// TwinCAT 3 PLC project PRG_B_Base
// Title: B_Base
// Company: RafalOS
// Author: Rafał Osajda
// ProjectVersion: 0.0.0.59
// ProgramVersion: 3.1.4024.0
// libraries:
//   Tc2_Standard, * (Beckhoff Automation GmbH)
//   Tc2_System, * (Beckhoff Automation GmbH)
//   Tc2_Utilities, * (Beckhoff Automation GmbH)
//   Tc3_Module, * (Beckhoff Automation GmbH)
// project tree:
//   DUTs Events/ E_BaseEvents_Category.TcDUT (not stored), E_BaseEvents_Action.TcDUT, ST_BaseEvents.TcDUT, ST_BaseEvents_ActiveEvents.TcDUT, ST_BaseEvents_Definition.TcDUT, ST_BaseEvents_Queue.TcDUT, ST_BaseEvents_Memory.TcDUT, ST_BaseEvents_RowInQueue.TcDUT, ST_BaseEvents_RowInMemory.TcDUT, ST_BaseEvents_InformationAboutEventsForHMI.TcDUT
//   DUTs/ E_BaseElementType.TcDUT, E_BaseLocation.TcDUT, E_BaseMachineState.TcDUT, E_BaseMachineMode.TcDUT, ST_BaseCommonData.TcDUT (not stored), ST_BaseDescriptor.TcDUT (not stored), ST_BaseElementIdentifier.TcDUT, ST_BaseLocationDesctription.TcDUT, ST_BaseLabel.TcDUT
//   FUNs/ CreateElementCode.TcPOU
//   GVLs/ GVL_BaseConstans.TcGVL
//   ITFs/ ITF_DecoratedElement.TcIO
//   / PlcTask.TcTTO (not stored)
//   POUs Compilation/ PRG_Compilation.TcPOU
//   POUs/A01_Base/ ITF_Base.TcIO (not stored), FB_Base.TcPOU
//   POUs/A07_FB_BaseTopElement/ ITF_BaseSaM.TcIO, ITF_BaseSaMStateMethod.TcIO, FB_BaseTopElement.TcPOU, ITF_BaseTopElement.TcIO, ITF_BaseTopElement_HMI_Connector.TcIO
//   POUs/B01_Komunikator/ ITF_BaseCommunicator.TcIO, ITF_BaseMessengerRecipient.TcIO (not stored), ITF_BaseMessengerSender.TcIO, FB_BaseCommunicator.TcPOU, ST_BaseCommunicatorData.TcDUT (not stored), ST_BaseCommunicatorStack.TcDUT (not stored), ST_BaseCommunicatorMassege.TcDUT
//   POUs/B02_Recipes/ FB_BaseRecipe.TcPOU, ITF_BaseCreateTemplateOfRecipe.TcIO, ITF_BaseCreatingTemplateMethod.TcIO, ST_BaseRecipeListRow.TcDUT (not stored), ST_BaseRecipe.TcDUT
//   POUs/A00_Basic/ FB_BaseLabel.TcPOU, FB_BaseTime.TcPOU, FB_BaseCommand.TcPOU, FB_BaseDescriptor.TcPOU, FB_BaseFlag.TcPOU, FB_BaseImpulse.TcPOU, FB_BaseLocation.TcPOU, ITF_BaseDescriptor.TcIO, ITF_BaseFlag.TcIO, ITF_BaseFlagGet.TcIO (not stored), ITF_BaseFlagSet.TcIO, ITF_BaseImpulse.TcIO, ITF_BaseLabel.TcIO (not stored), ITF_BaseLocation.TcIO, ITF_BaseTime.TcIO
//   POUs/A02_FB_BaseLogger/ FB_BaseLogger.TcPOU, ITF_BaseLogger.TcIO, ITF_BaseLogger_HMI_Connector.TcIO, ITF_BaseLogger_Item.TcIO, ST_BaseLogger_ItemDataToDisplay.TcDUT
//   POUs/A03_FB_BaseLoggerElement/ FB_BaseLoggerElement.TcPOU, ITF_BaseLoggerElement.TcIO, ITF_BaseLoggerElement_HMI_Connector.TcIO
//   POUs/A04_FB_BaseComponent/ FB_BaseComponent.TcPOU, ITF_BaseComponent.TcIO, ITF_BaseComponent_HMI_Connector.TcIO, ST_Parameters.TcDUT (not stored)
//   POUs/A05_FB_BaseControlElement/ FB_BaseControlElement.TcPOU, ITF_BaseControlElement.TcIO, ITF_BaseControlElement_HMI_Connector.TcIO (not stored), ST_BaseControlElement_Power.TcDUT (not stored), ST_BaseControlElement_Homing.TcDUT
//   POUs/A06_FB_BaseGroupElement/ FB_BaseGroupElement.TcPOU, ITF_BaseGroupElement.TcIO, ITF_BaseGroupElement_HMI_Connector.TcIO
// real-time tasks:
//   TASK PlcTask: cycle T#10ms, priority 20, ADS port 350

// ---- DUTs Events/E_BaseEvents_Action.TcDUT
{attribute 'qualified_only'}
{attribute 'strict'}
{attribute 'to_string'}
TYPE E_BaseEvents_Action :
(
	Start 		:= 0,
	Stop		:= 1,
	Confirm		:= 2
);
END_TYPE

// ---- DUTs Events/ST_BaseEvents.TcDUT
TYPE ST_BaseEvents :
STRUCT
	uiNumberOfAdded					: UINT;	//Iloscdodanych zgloszen
	
	arrDefinitions					: ARRAY [1..GVL_BaseConstans.MAX_EVENTS_PER_ITEM] OF ST_BaseEvents_Definition;
	arrState						: ARRAY [1..GVL_BaseConstans.MAX_EVENTS_PER_ITEM] OF BOOL;
	arrConfirmation					: ARRAY [1..GVL_BaseConstans.MAX_EVENTS_PER_ITEM] OF BOOL;

	iNumberOfActiveEvents			: INT; //zmienna pomocnicza informująca o ilości wszystkich aktywnych zgłoszeń

	bLoggerDataCompleted			: BOOL;
END_STRUCT
END_TYPE

// ---- DUTs Events/ST_BaseEvents_ActiveEvents.TcDUT
TYPE ST_BaseEvents_ActiveEvents :
STRUCT
	bIsActive						: BOOL;	//informacja o wszysktkich aktywnych zgloszeniach
	iNumberOfActive					: INT;
	iTotalNumer						: INT;	//ilosc wszystkich zgloszonych zgloszen
	bIsActiveWithConfirmation		: BOOL;	//infdormacja o aktywnych bledach ktore wymagaja potwierdzenia
	iNumberOfActiveWithConfirmation	: INT;	//ilosc wszystkich zdarzen do potwierdzenia
	arrNumberOfActive				: ARRAY [0..GVL_BaseConstans.NUMBER_OF_EVENT_CATEGORIES] OF INT;	//ilosc wszystkich aktywnych zgloszen z podziałem na rodzaje
	arrTotalNumer					: ARRAY [0..GVL_BaseConstans.NUMBER_OF_EVENT_CATEGORIES] OF INT;	//ilosc wszystkich zgloszonych z podzialem na rodzaje
	arrActive						: ARRAY [0..GVL_BaseConstans.NUMBER_OF_EVENT_CATEGORIES] OF BOOL; 	//informacja który z rodzajów zgłoszęń jest aktywny
END_STRUCT
END_TYPE

// ---- DUTs Events/ST_BaseEvents_Definition.TcDUT
TYPE ST_BaseEvents_Definition :
STRUCT
	uiID									: UINT;						//unikalny numer zgloszenia dla całego projektu nadawany automatycznie 
	uiIDWElemencie							: UINT;						//unikalny numer w elemencie - ustawiany podczas dodawania zgłoszenia DO elementu
	bIgnorujPowtorzenia						: BOOL;						//jak true nie zliczaj powtorzeń wystapienia np komunikaty - alarmy 
	uiLicznikPowtorzen						: UINT;						//licznik powtórzeń po którym ma się zgłosic błąd
	eRodzajZdarzenia						: E_BaseEvents_Category;			//BYTE;	//1 - blad, 2 - ostrzezenie, 3 - wiadomosc, 4 - safety
	stOpis									: ST_BaseLabel;
	bWymagaPotwierdzenia					: BOOL;						// w przypadków niektórych zgłoszeń żeby błąd został skasowany należy go zatwierdzić że operator go zobaczył
END_STRUCT
END_TYPE

// ---- DUTs Events/ST_BaseEvents_Queue.TcDUT
TYPE ST_BaseEvents_Queue :
STRUCT
	arrEvents						: ARRAY [1..GVL_BaseConstans.MAX_NUMBER_OF_EVENTS_IN_THE_QUEUE] OF ST_BaseEvents_RowInQueue;
	iNumerOfEvents					: INT;
	bChangeInMemory					: BOOL;		//informacja dla wyświetlania żeby odświerzyć
	
END_STRUCT
END_TYPE

// ---- DUTs Events/ST_BaseEvents_Memory.TcDUT
TYPE ST_BaseEvents_Memory :
STRUCT
	arrRow						: ARRAY [1..GVL_BaseConstans.MAX_NUMBER_EVENTS_IN_MEMORY] OF ST_BaseEvents_RowInMemory;
	iNumberOfRow				: INT;
	
END_STRUCT
END_TYPE

// ---- DUTs Events/ST_BaseEvents_RowInQueue.TcDUT
TYPE ST_BaseEvents_RowInQueue :
STRUCT
	uiIDEvent								: UINT;					//unikalny numer zgloszenia dla całego projektu nadawany automatycznie 
	uiIDItem								: UINT;					// unikalny numer elementu w systemie
	bActive									: BOOL;             	
	bIgnoreRepetitions						: BOOL;					//jak true nie zliczaj powtorzeń wystapienia np komunikaty
	uiRepetitionCounter						: UINT;             	
	dtStart									: DT;					//poczatek wystepowania zgłoszenia
	dtFinish								: DT;					//koniec wystepowaniazgloszenia
	dtConfirmed								: DT;					// stempel potwierdzenia 
	bConfirm								: BOOL;					//informacja czy bo byc zgłoszenie potwierdzone
	eEventCategory							: E_BaseEvents_Category;
	eEventAction							: E_BaseEvents_Action;	//okresla rodzaj zgloszenia w kolejce Start stop 
END_STRUCT
END_TYPE

// ---- DUTs Events/ST_BaseEvents_RowInMemory.TcDUT
TYPE ST_BaseEvents_RowInMemory :
STRUCT
	uiIDEvent								: UINT;				//unikalny numer zgloszenia dla całego projektu nadawany automatycznie 
	uiIDItem								: UINT;				// unikalny numer elementu w systemie
	bActive									: BOOL;
	bIgnoreRepetitions						: BOOL;				//jak true nie zliczaj powtorzeń wystapienia np komunikaty
	uiRepetitionCounter						: UINT;
	dtStart									: DT;				//poczatek wystepowania zgłoszenia
	dtFinish								: DT;				//koniec wystepowaniazgloszenia
	dtConfirmed								: DT;				// stempel potwierdzenia 
	bConfirm								: BOOL;				//informacja czy potrzebne jest potwierdzenie 
	bConfirmed								: BOOL;				//pamięta czy już potwierdzone
	eEventCategory							: E_BaseEvents_Category;
END_STRUCT
END_TYPE

// ---- DUTs Events/ST_BaseEvents_InformationAboutEventsForHMI.TcDUT
(*			
	EVERDE sp. z o.o.
	Rafał Osajda		03.09.2025		TC 4024.66
	Informacja czy w danym elemencie jest jakieś nowe zgłoszenie jeszcze nei wyświetlane i ilosc zgloszen calkowita
*)
TYPE ST_BaseEvents_InformationAboutEventsForHMI :
STRUCT
	bNew				: BOOL;	//nowe
	iQuantity			: INT;	//Ilość
END_STRUCT
END_TYPE

// ---- DUTs/E_BaseElementType.TcDUT
{attribute 'qualified_only'}
{attribute 'strict'}
TYPE E_BaseElementType :
(
	eComponent 	:= 1,
	eControl	:= 2,
	eGroup		:= 3,
	eTop		:= 4
);
END_TYPE

// ---- DUTs/E_BaseLocation.TcDUT
{attribute 'qualified_only'}
{attribute 'strict'}
{attribute 'to_string'}
TYPE E_BaseLocation :
(
	pl		:= 1,
	en		:= 2,
	de		:= 3
);
END_TYPE

// ---- DUTs/E_BaseMachineState.TcDUT
{attribute 'qualified_only'}
{attribute 'strict'}
TYPE E_BaseMachineState :
(
	Undefined     						:= 0,
	Aborting      						:= 1,
	Aborted       						:= 2,
	Clearing      						:= 3,
	Stopping      						:= 4,
	Stopped       						:= 5,
	Resetting     						:= 6,
	Idle          						:= 7,
	Starting      						:= 8,
	Execute       						:= 9,
	Suspending    						:= 10,
	Suspended     						:= 11,
	Unsuspending  						:= 12,
	Holding       						:= 13,
	Held          						:= 14,
	Unholding     						:= 15,
	Completing    						:= 16,
	Complete      						:= 17
);
END_TYPE

// ---- DUTs/E_BaseMachineMode.TcDUT
{attribute 'qualified_only'}
{attribute 'strict'}
TYPE E_BaseMachineMode :
(
    NotAllowed			:= 0,
    Production			:= 1,
    Maintenance			:= 2,
    Manual				:= 3,
    Washing				:= 4,
    Diagnostics			:= 5
//    Uzytkownika1		:= 6,
//    Uzytkownika2		:= 7,
//    Uzytkownika3		:= 8,
//    Uzytkownika4		:= 9	
);
END_TYPE

// ---- DUTs/ST_BaseElementIdentifier.TcDUT
{attribute 'global_init_slot' := '40501'} 
TYPE ST_BaseElementIdentifier :
STRUCT
	stName					: ST_BaseLabel;
	sCode					: STRING;		//unikalny kod elementu w postaci X.X.X
	uiID					: UINT;			//unikalny numer elementu
	eType					: E_BaseElementType;
END_STRUCT
END_TYPE

// ---- DUTs/ST_BaseLocationDesctription.TcDUT
TYPE ST_BaseLocationDesctription :
STRUCT
	wsDescription		: WSTRING;
	sCade				: STRING;
END_STRUCT
END_TYPE

// ---- DUTs/ST_BaseLabel.TcDUT
TYPE ST_BaseLabel :
STRUCT
	arrText		: ARRAY [1..GVL_BaseConstans.NUMBER_OF_LOCACIONS] OF WSTRING;
	
END_STRUCT
END_TYPE

// ---- POUs/B01_Komunikator/ST_BaseCommunicatorMassege.TcDUT
TYPE ST_BaseCommunicatorMassege :
STRUCT
	sText				: STRING;
	bToPickUp			: BOOL;		//informacja ze komunikat jest aktualny, po odebraniu przez odbiorce flaga znika
	bValue				: BOOL;
	rValue				: REAL;
END_STRUCT
END_TYPE

// ---- POUs/A02_FB_BaseLogger/ST_BaseLogger_ItemDataToDisplay.TcDUT
TYPE ST_BaseLogger_ItemDataToDisplay :
STRUCT
	sCode						: STRING;
	sEventCategory				: STRING;
	eEventCategory				: E_BaseEvents_Category;
	stDescription				: ST_BaseLabel;
	stItemName					: ST_BaseLabel;
END_STRUCT
END_TYPE

// ---- POUs/A05_FB_BaseControlElement/ST_BaseControlElement_Homing.TcDUT
TYPE ST_BaseControlElement_Homing :
STRUCT
	cmdExecute				: FB_BaseCommand;
	bIsNeeded				: BOOL := TRUE;		//pamieta czy juz element został wybazowany na początku true po bazowaniu zostaje ustawione na false
	bWithoutHoming			: BOOL;				//ustawienie czy ma być bazowanie czy nie
	iElementHomingStep		: INT;				//krok dla elementów złożonych biblioteki
	iChildHomingStep		: int;				//krok dla metody bazowania wykorzystywany w potomkach FB
END_STRUCT
END_TYPE

// ---- POUs/B02_Recipes/ST_BaseRecipe.TcDUT
TYPE ST_BaseRecipe :
STRUCT
	arrIngredient			: ARRAY [1..GVL_BaseConstans.MAX_NUMBER_Of_INGREDIENTS] OF ST_BaseDescriptor;
	uiNumber				: UINT;	//ilosc dodanych skladnikow
	stTexts					: ST_BaseLabel;
	uiTemplate				: UINT;	//określenie z którego szablonu stworzona receptura różna programy Wykonawcze
END_STRUCT
END_TYPE

// ---- GVLs/GVL_BaseConstans.TcGVL
{attribute 'qualified_only'}
{attribute 'global_init_slot' := '40502'} 
VAR_GLOBAL CONSTANT
	(*	Ogólne		*)
	FINISH_STEP								: INT := 1000;

	(* Lokalizacje	*)
	NUMBER_OF_LOCATIONS						: INT := 3;		//Ilość obsługiwanych języków w systemi

	(*	Loger		*)
	MAX_NUMBER_OF_EVENTS_IN_THE_QUEUE		: UINT := 20;	//rozmiar kolejki 
	MAX_EVENTS_PER_ITEM						: UINT := 50;	//maksymalna ilosc zgłoszeń dla jednego elementu
	MAX_EVENTS_IN_MEMORY					: UINT := 500;	//ilość pamiętanych zgłoszeń
	NUMBER_OF_EVENT_CATEGORIES				: INT := 4;
	MAX_EVENTS_TO_SHOW						: INT := 100;	//ilośc elementów które będą wyświetlane

	(*	Receptury	*)
	MAX_NUMBER_Of_INGREDIENTS				: UINT := 400;// Parametry.MAX_ILOSC_SKLADNIKOW;
	MAX_NUMBER_OF_TEMPLATES					: UINT := 5;// Parametry.MAX_ILOSC_SZABLONOW;
	MAX_NUMBER_OF_RECIPES					: UINT := 10;// Parametry.MAX_ILOSC_RECEPTUR;

	(*	Parametry	*)
	MAX_NUMBER_OF_PARAMETERS				: INT := 100;

	(*	Komponenty i Elementy	*)
	MAX_NUMBER_OF_ALL_ITEM					: UINT := 500;	// liczba wszystkich komponentów we wszystkich podzespolach bazowych
	MAX_ITEM_PER_ELEMENT					: UINT := 150;
	MAX_NUMBER_OF_TOP_ELEMENT				: UINT := 10;
	MAX_NESTING_LEVEL						: UINT	:= 5;	//ilość zagnieżdzonych elementów liczone z topelement

	(*	Komunikator		*)
	MAX_NUMBER_OF_CLIENTS					: INT := 20;
	MAX_NUMBER_OF_MASSAGES					: INT := 200;
	MAX_NUMBER_OF_MASSAGES_ON_STACK			: INT := 200;
	
END_VAR

// ---- ITFs/ITF_DecoratedElement.TcIO
INTERFACE ITF_DecoratedElement

METHOD GetITFComponent : ITF_BaseComponent
VAR_INPUT
END_VAR
END_METHOD

METHOD GetITFControlElement : ITF_BaseControlElement
VAR_INPUT
END_VAR
END_METHOD

METHOD GetITFGroupElement : ITF_BaseGroupElement
VAR_INPUT
END_VAR
END_METHOD

METHOD GetITFLoggerElement : ITF_BaseLoggerElement
VAR_INPUT
END_VAR
END_METHOD

METHOD GetITFTopElement : ITF_BaseTopElement
VAR_INPUT
END_VAR
END_METHOD

END_INTERFACE

// ---- POUs/A07_FB_BaseTopElement/ITF_BaseSaM.TcIO
INTERFACE ITF_BaseSaM

METHOD PUBLIC GetMode : E_BaseMachineMode
VAR_INPUT
END_VAR
END_METHOD

METHOD PUBLIC GetState : E_BaseMachineState
VAR_INPUT
END_VAR
END_METHOD

(*			
	EVERDE sp. z o.o.
	Rafał Osajda		25.10.2025		TC 4024.66
	Czy trwa zmianay trybu
*)
METHOD PUBLIC IsChangeModeBusy : BOOL
VAR_INPUT
END_VAR
END_METHOD

(*			
	EVERDE sp. z o.o.
	Rafał Osajda		25.10.2025		TC 4024.66
	Czy trwa zmiana stanu
*)
METHOD PUBLIC IsChangeStateBusy : BOOL
VAR_INPUT

END_VAR
END_METHOD

END_INTERFACE

// ---- POUs/A07_FB_BaseTopElement/ITF_BaseSaMStateMethod.TcIO
INTERFACE ITF_BaseSaMStateMethod

(*			RafalOS
	Rafał Osajda		27.10.2024		TC 4026.11		wer. 0.0.0.1
	metoda obsługi czekania na reset
*)
METHOD SP_Aborted : BOOL
END_METHOD

(*			RafalOS
	Rafał Osajda		27.10.2024		TC 4026.11		wer. 0.0.0.1
	metoda obsługi wyłączania napędów po wciśnięciu grzyba
*)
METHOD SP_Aborting : BOOL
END_METHOD

(*			RafalOS
	Rafał Osajda		27.10.2024		TC 4026.11		wer. 0.0.0.1
	metoda obsługi czyszczenia po grzybie
*)
METHOD SP_Clearing : BOOL
END_METHOD

(*			RafalOS
	Rafał Osajda		27.10.2024		TC 4026.11		wer. 0.0.0.1
	metoda obsługi Wykonania określonego zadania
*)
METHOD SP_Complete : BOOL
END_METHOD

(*			RafalOS
	Rafał Osajda		27.10.2024		TC 4026.11		wer. 0.0.0.1
	metoda obsługi pracy automatycznej do zadanej wartości ilości elementów
*)
METHOD SP_Completing : BOOL
END_METHOD

(*			RafalOS
	Rafał Osajda		27.10.2024		TC 4026.11		wer. 0.0.0.1
	metoda obsługi pracy
*)
METHOD SP_Execute : BOOL
END_METHOD

(*			RafalOS
	Rafał Osajda		27.10.2024		TC 4026.11		wer. 0.0.0.1
	metoda obsługi wstrzymania pracy ze względów na błędy/alarmy
*)
METHOD SP_Held : BOOL
END_METHOD

(*			RafalOS
	Rafał Osajda		27.10.2024		TC 4026.11		wer. 0.0.0.1
	metoda obsługi wyjścia z wstrzymania pracy
*)
METHOD SP_Holding : BOOL
END_METHOD

(*			RafalOS
	Rafał Osajda		27.10.2024		TC 4026.11		wer. 0.0.0.1
	metoda obsługi czekania na dalsze rozkazy
*)
METHOD SP_Idle : BOOL
END_METHOD

(*			RafalOS
	Rafał Osajda		27.10.2024		TC 4026.11		wer. 0.0.0.1
	Metoda sprawdzająca czy elementy maszyny ustawiły się na 0 wczytanie parametrów pracy
*)
METHOD SP_Resetting : BOOL
END_METHOD

(*			RafalOS
	Rafał Osajda		27.10.2024		TC 4026.11		wer. 0.0.0.1
	metoda obsługi uruchamiania pracy
*)
METHOD SP_Starting : BOOL
END_METHOD

(*			RafalOS
	Rafał Osajda		27.10.2024		TC 4026.11		wer. 0.0.0.1
	metoda obsługi czekania na dalsze rozkazy
*)
METHOD SP_Stopped : BOOL
END_METHOD

(*			RafalOS
	Rafał Osajda		27.10.2024		TC 4026.11		wer. 0.0.0.1
	Metoda sprawdzająca czy wszystkie operacje zostały już zakończone i można wyłaczyc pracę 
*)
METHOD SP_Stopping : BOOL
END_METHOD

(*			RafalOS
	Rafał Osajda		27.10.2024		TC 4026.11		wer. 0.0.0.1
	metoda obsługi wstrzymania pracy ze względu na warunki zewnętrzne np brak materialu
*)
METHOD SP_Suspended : BOOL
END_METHOD

(*			RafalOS
	Rafał Osajda		27.10.2024		TC 4026.11		wer. 0.0.0.1
	metoda obsługi zawieszania pracy ze wzgledu na okoliczności zewnętrzne
*)
METHOD SP_Suspending : BOOL
END_METHOD

(*			RafalOS
	Rafał Osajda		27.10.2024		TC 4026.11		wer. 0.0.0.1
	metoda obsługi stanu zabroniownego - występuje tylko przy starcie
*)
METHOD SP_Undefined : BOOL
END_METHOD

(*			RafalOS
	Rafał Osajda		27.10.2024		TC 4026.11		wer. 0.0.0.1
	metoda obsługi uruchamiania po wstrzymaniu
*)
METHOD SP_Unholding : BOOL
END_METHOD

(*			RafalOS
	Rafał Osajda		27.10.2024		TC 4026.11		wer. 0.0.0.1
	metoda obsługi uruchamiania po wstzryamaniu
*)
METHOD SP_Unsuspending : BOOL
END_METHOD

END_INTERFACE

// ---- POUs/B01_Komunikator/ITF_BaseCommunicator.TcIO
INTERFACE ITF_BaseCommunicator

METHOD PUBLIC ReceiveData_BOOL : BOOL
VAR_INPUT
	sText			: STRING;
	itfRecipient	: ITF_BaseMessengerRecipient;
END_VAR
VAR_OUTPUT
	bValue			: BOOL;	
END_VAR
END_METHOD

METHOD PUBLIC ReceiveData_REAL : BOOL
VAR_INPUT
	sText			: STRING;
	itfRecipient	: ITF_BaseMessengerRecipient;
END_VAR
VAR_OUTPUT
	rValue			: REAL;	
END_VAR
END_METHOD

(*			
	EVERDE sp. z o.o.
	Rafał Osajda		30.07.2025		TC 4024.66
	Wysyła potwierdzenie że odebrał dane
*)
METHOD PUBLIC ReceiveDataConfirm : BOOL
VAR_INPUT
	sText				: STRING;
	itfRecipient		: ITF_BaseMessengerRecipient;
END_VAR
END_METHOD

METHOD SendData_BOOL : BOOL
VAR_INPUT
	sText		: STRING;
	itfSender	: ITF_BaseMessengerSender;
END_VAR
END_METHOD

METHOD SendData_REAL : BOOL
VAR_INPUT
	sText		: STRING;
	rValue		: REAL;
	itfSender	: ITF_BaseMessengerSender;
END_VAR
END_METHOD

END_INTERFACE

// ---- POUs/B01_Komunikator/ITF_BaseMessengerSender.TcIO
INTERFACE ITF_BaseMessengerSender

END_INTERFACE

// ---- POUs/A00_Basic/ITF_BaseDescriptor.TcIO
INTERFACE ITF_BaseDescriptor

END_INTERFACE

// ---- POUs/A00_Basic/ITF_BaseFlag.TcIO
INTERFACE ITF_BaseFlag extends ITF_BaseFlagGet, ITF_BaseFlagSet

END_INTERFACE

// ---- POUs/A00_Basic/ITF_BaseFlagSet.TcIO
INTERFACE ITF_BaseFlagSet

METHOD PUBLIC SetFlag
VAR_INPUT
	bState				: BOOL;
END_VAR
END_METHOD

END_INTERFACE

// ---- POUs/A00_Basic/ITF_BaseImpulse.TcIO
INTERFACE ITF_BaseImpulse

END_INTERFACE

// ---- POUs/A00_Basic/ITF_BaseLocation.TcIO
INTERFACE ITF_BaseLocation

END_INTERFACE

// ---- POUs/A00_Basic/ITF_BaseTime.TcIO
INTERFACE ITF_BaseTime

(*			
	EVERDE sp. z o.o.
	Rafał Osajda		01.09.2025		TC 4024.66
	Konwetrtuje DT to string do postaci DD/MM/YYYY GG:MM:SS
*)
METHOD PUBLIC BaseDTToString : STRING
VAR_INPUT
	inDT					: DT;
END_VAR
END_METHOD

(*			
	EVERDE sp. z o.o.
	Rafał Osajda		01.09.2025		TC 4024.66
	Konwetrtuje DT to string do postaci DD_MM_YYYY GG_MM_SS - wersja do nazywania plików logów
*)
METHOD PUBLIC BaseDTToString_ : STRING
VAR_INPUT
	inDT				: DT;
END_VAR
END_METHOD

(*			
	EVERDE sp. z o.o.
	Rafał Osajda		01.09.2025		TC 4024.66
	Konwertuje czas LTIME do stringa z możliwością wyłączenia milisekund
*)
METHOD PUBLIC BaseLTimeToString : STRING
VAR_INPUT
	ltTime				: LTIME;
	bShowMS			: BOOL;
END_VAR
END_METHOD

(*			
	EVERDE sp. z o.o.
	Rafał Osajda		01.09.2025		TC 4024.66
	Konwertuje czas LTIME do stringa z możliwością wybrnia co ma być pokazywane do postaci DDDd:GG:MM:SS:MS
	dni nie rodziala na miesiące i lata 
*)
METHOD PUBLIC BaseLTimeToString_WhatShow : STRING
VAR_INPUT
	ltTime				: LTIME;
	bSwahDays			: BOOL;
	bShowHours			: BOOL;
	bShowMinutes		: BOOL;
	bShowSeconds		: BOOL;
	bShowMS				: BOOL;
END_VAR
END_METHOD

METHOD PUBLIC StampDT : DT
VAR_INPUT
END_VAR
END_METHOD

END_INTERFACE

// ---- POUs/A02_FB_BaseLogger/ITF_BaseLogger.TcIO
INTERFACE ITF_BaseLogger

METHOD PUBLIC AddItem : INT
VAR_INPUT
	itfItem				: ITF_BaseLogger_Item;
END_VAR
END_METHOD

METHOD PUBLIC ReportEvent : BOOL
VAR_INPUT
	stEvent					: ST_BaseEvents_RowInQueue;
END_VAR
END_METHOD

END_INTERFACE

// ---- POUs/A02_FB_BaseLogger/ITF_BaseLogger_HMI_Connector.TcIO
INTERFACE ITF_BaseLogger_HMI_Connector

(*			
	RafalOS
	Rafał Osajda		02.10.2025		TC 4024.66
	Zwraca czy nastąpiła jakaś zmiana w pamięci zgłoszeń - całej nie tylko dla jakiegoś elementu
*)
METHOD PUBLIC GetChangeInMemory : BOOL
VAR_INPUT
END_VAR
END_METHOD

METHOD PUBLIC GetEventCounts : ST_BaseEvents_ActiveEvents
VAR_INPUT
END_VAR
END_METHOD

METHOD PUBLIC GetEventCountsForItem : ST_BaseEvents_ActiveEvents
VAR_INPUT
	uiIDItem: UINT;
END_VAR
END_METHOD

METHOD PUBLIC GetInformationFromItem : ST_BaseLogger_ItemDataToDisplay
VAR_INPUT
	uiIDItem				: UINT;
	uiIDEvent				: UINT;
END_VAR
END_METHOD

METHOD GetReferenceToStmemory : REFERENCE TO ST_BaseEvents_Memory
VAR_INPUT
	
END_VAR
END_METHOD

(*			
	RafalOS
	Rafał Osajda		02.10.2025		TC 4024.66
	
*)
METHOD PUBLIC ResetChangeInMemory : BOOL
VAR_INPUT
END_VAR
END_METHOD

END_INTERFACE

// ---- POUs/A02_FB_BaseLogger/ITF_BaseLogger_Item.TcIO
INTERFACE ITF_BaseLogger_Item

METHOD GetInformationToDisplayEvent : ST_BaseLogger_ItemDataToDisplay
VAR_INPUT
	uiIDEvent				: UINT;
END_VAR
END_METHOD

END_INTERFACE

// ---- POUs/A03_FB_BaseLoggerElement/ITF_BaseLoggerElement.TcIO
INTERFACE ITF_BaseLoggerElement EXTENDS ITF_Base

(*			
	EVERDE sp. z o.o.
	Rafał Osajda		24.03.2025		TC 4024.66
	Definicja nowego zgłoszenia
*)
METHOD PUBLIC EventsDefinition : BOOL
END_METHOD

METHOD PUBLIC GetCode : STRING
VAR_INPUT
END_VAR
END_METHOD

METHOD PUBLIC GetID : UINT
VAR_INPUT
END_VAR
END_METHOD

METHOD PUBLIC GetIdentyfier : ST_BaseElementIdentifier
VAR_INPUT
END_VAR
END_METHOD

METHOD PUBLIC GetName : ST_BaseLabel
VAR_INPUT
END_VAR
END_METHOD

METHOD PUBLIC GetType : E_BaseElementType
VAR_INPUT
END_VAR
END_METHOD

METHOD PUBLIC SetCode
VAR_INPUT
	sCode							: STRING;
	sAdd							: STRING;
END_VAR
END_METHOD

(*			
	EVERDE sp. z o.o.
	Rafał Osajda		03.10.2025		TC 4024.66
	nadawanie unikalnych ID dla zdarzeń
*)
METHOD PUBLIC SetEventsIDs : UINT
VAR_INPUT
	uiNewID		: UINT;
END_VAR
END_METHOD

METHOD PUBLIC SetID : UINT
VAR_INPUT
	uiID					: UINT;
END_VAR
END_METHOD

METHOD PUBLIC SetName
VAR_INPUT
	stName				: ST_BaseLabel;
END_VAR
END_METHOD

METHOD PUBLIC SetType
VAR_INPUT
	eType					: E_BaseElementType;
END_VAR
END_METHOD

END_INTERFACE

// ---- POUs/A03_FB_BaseLoggerElement/ITF_BaseLoggerElement_HMI_Connector.TcIO
INTERFACE ITF_BaseLoggerElement_HMI_Connector

(*			
	EVERDE sp. z o.o.
	Rafał Osajda		09.06.2025		TC 4024.66
	Szuka czy ma zgłoszenie i zadanym ID jak tak to usuwa i zwraca true w przeciwnym razie zwraca false 
*)
METHOD PUBLIC EventAcknowledgeByID : BOOL
VAR_INPUT
	uiIDEvent				: UINT;
END_VAR
END_METHOD

(*			
	EVERDE sp. z o.o.
	Rafał Osajda		09.06.2025		TC 4024.66
	Szuka czy ma zgłoszenie i zadanym ID jak tak to usuwa i zwraca true w przeciwnym razie zwraca false 
*)
METHOD PUBLIC EventSetInactiveByID : BOOL
VAR_INPUT
	uiIDEvent				: UINT;
END_VAR
END_METHOD

METHOD PUBLIC GetCode : STRING
VAR_INPUT
END_VAR
END_METHOD

METHOD PUBLIC GetID : UINT
VAR_INPUT
END_VAR
END_METHOD

METHOD PUBLIC GetIdentyfier : ST_BaseElementIdentifier
VAR_INPUT
END_VAR
END_METHOD

METHOD PUBLIC GetName : ST_BaseLabel
VAR_INPUT
END_VAR
END_METHOD

METHOD PUBLIC GetType : E_BaseElementType
VAR_INPUT
END_VAR
END_METHOD

END_INTERFACE

// ---- POUs/A04_FB_BaseComponent/ITF_BaseComponent.TcIO
INTERFACE ITF_BaseComponent EXTENDS ITF_BaseLoggerElement

(*			
	EVERDE sp. z o.o.
	Rafał Osajda		27.03.2025		TC 4024.66
	Obsluga bledow sprawdzanie czy jakis blad sie nei pojawil i ustawienie stanu lub wylaczenie
*)
METHOD PUBLIC ExecuteEveryCycle_Error
VAR_INPUT
END_VAR
END_METHOD

(*			
	EVERDE sp. z o.o.
	Rafał Osajda		27.03.2025		TC 4024.66
	Wywolanie co cykl operacji 
*)
METHOD PUBLIC ExecuteEveryCycle_Operation
VAR_INPUT
END_VAR
END_METHOD

(*			
	EVERDE sp. z o.o.
	Rafał Osajda		27.03.2025		TC 4024.66
	Aktualizacja flag 
*)
METHOD PUBLIC ExecuteEveryCycle_Status
VAR_INST
END_VAR
END_METHOD

(*			
	EVERDE sp. z o.o.
	Rafał Osajda		27.03.2025		TC 4024.66
	Testowanie czy nei pojawil sie jakis rozkaz i uruchomienie odpowiednich operacji
*)
METHOD PUBLIC ExecuteEveryCycle_Test
VAR_INPUT
END_VAR
END_METHOD

METHOD PUBLIC FirstCycle : BOOL
VAR_INPUT
END_VAR
END_METHOD

METHOD PUBLIC IsValidCommonData : BOOL
VAR_INPUT
END_VAR
END_METHOD

(*			
	EVERDE sp. z o.o.
	Rafał Osajda		07.10.2025		TC 4024.66
	Dodpisywanie się do listy logera
*)
METHOD PUBLIC JoinTheLogger : BOOL
VAR_INPUT
END_VAR
END_METHOD

METHOD PUBLIC LinkCommonData : BOOL
VAR_INPUT
	stCommonData				: REFERENCE TO ST_BaseCommonData;
END_VAR
END_METHOD

(*			
	EVERDE sp. z o.o.
	Rafał Osajda		26.03.2025		TC 4024.66
	Dodawanie parametru do elementu wykonawczego - metode wywołać przy pierwszym uruchomieniu programu by wgrać parametry do pamięci
	później używać tylko edycji lub przywracania wartości domyślnych
*)
METHOD PUBLIC ParameterAdd : BOOL
VAR_INPUT
	stParameter			: ST_BaseDescriptor;
END_VAR
END_METHOD

(*			
	EVERDE sp. z o.o.
	Rafał Osajda		26.03.2025		TC 4024.66
	Modyfikuje wartość domyślną w istniejącym parametrze - true jak się zmiana udała
*)
METHOD PUBLIC ParameterCorrectDefaultValue : BOOL
VAR_INPUT
	uiNumber			: UINT;
	rValue				: REAL;
END_VAR
END_METHOD

METHOD PUBLIC ParameterCorrectName : BOOL
VAR_INPUT
	eLocation					: E_BaseLocation;
	uiNumberOfParameter			: UINT;
	wsDescription				: WSTRING;
END_VAR
END_METHOD

(*			
	EVERDE sp. z o.o.
	Rafał Osajda		26.03.2025		TC 4024.66
	Modyfikuje wartość w istniejącym parametrze - true jak się zmiana udała
*)
METHOD PUBLIC ParameterCorrectValue : BOOL
VAR_INPUT
	uiNumber			: UINT;
	rValue				: REAL;
END_VAR
END_METHOD

METHOD PUBLIC ParameterGet : ST_BaseDescriptor
VAR_INPUT
	uiNumer				: UINT;
END_VAR
END_METHOD

(*			
	EVERDE sp. z o.o.
	Rafał Osajda		26.03.2025		TC 4024.66
	Zwraca wartosc domyslna
*)
METHOD PUBLIC ParameterGetDefaultValue : REAL
VAR_INPUT
	uiNumber				: UINT;
END_VAR
END_METHOD

(*			
	EVERDE sp. z o.o.
	Rafał Osajda		26.03.2025		TC 4024.66
	Zwraca wartość MAX
*)
METHOD PUBLIC ParameterGetMax : REAL
VAR_INPUT
	uiNumber				: UINT;
END_VAR
END_METHOD

(*			
	EVERDE sp. z o.o.
	Rafał Osajda		26.03.2025		TC 4024.66
	Zwraca wartość MIN
*)
METHOD PUBLIC ParameterGetMin : REAL
VAR_INPUT
	uiNumber				: UINT;
END_VAR
END_METHOD

METHOD PUBLIC ParameterGetNumberOfAdded : UINT
VAR_INPUT
END_VAR
END_METHOD

(*			
	EVERDE sp. z o.o.
	Rafał Osajda		26.03.2025		TC 4024.66
	Zwraca jednostke
*)
METHOD PUBLIC ParameterGetUnit : STRING(6)
VAR_INPUT
	uiNumber				: uINT;
END_VAR
END_METHOD

(*			
	EVERDE sp. z o.o.
	Rafał Osajda		26.03.2025		TC 4024.66
	Zwraca wartość
*)
METHOD PUBLIC ParameterGetValue : REAL
VAR_INPUT
	uiNumber				: UINT;
END_VAR
END_METHOD

(*			
	EVERDE sp. z o.o.
	Rafał Osajda		26.03.2025		TC 4024.66
	Modyfikacja istniejącego parametra jako przypisanie nowego deskryptora
*)
METHOD PUBLIC ParameterModify : BOOL
VAR_INPUT
	uiNumber			: UINT;
	stParameter			: ST_BaseDescriptor;
END_VAR
END_METHOD

METHOD PUBLIC ParameterRestoreDefaultValue : BOOL
VAR_INPUT
	uiNumber		: UINT;
END_VAR
END_METHOD

(*			
	EVERDE sp. z o.o.
	Rafał Osajda		04.05.2025		TC 4024.66
	Skasowanie i utworzenie tablicy parametrów od nowa 
*)
METHOD PUBLIC ParametersCreate : BOOL
END_METHOD

(*			
	EVERDE sp. z o.o.
	Rafał Osajda		04.05.2025		TC 4024.66
	Przywrocenie parametrow - in na false to tylko ten element true razem z podelementami
*)
METHOD PUBLIC ParameterSetToDefault : BOOL
END_METHOD

METHOD PUBLIC Reset : BOOL
VAR_INPUT
END_VAR
END_METHOD

METHOD PUBLIC ResetGetBusy : BOOL
VAR_INPUT
END_VAR
END_METHOD

METHOD PUBLIC ResetGetStatus : BOOL
VAR_INPUT
END_VAR
END_METHOD

END_INTERFACE

// ---- POUs/A04_FB_BaseComponent/ITF_BaseComponent_HMI_Connector.TcIO
INTERFACE ITF_BaseComponent_HMI_Connector EXTENDS ITF_BaseLoggerElement_HMI_Connector

END_INTERFACE

// ---- POUs/A05_FB_BaseControlElement/ITF_BaseControlElement.TcIO
INTERFACE ITF_BaseControlElement EXTENDS ITF_BaseComponent

(*			
	EVERDE sp. z o.o.
	Rafał Osajda		31.03.2025		TC 4024.66
	Flaga że w tej sesji pracy maszyny element został już wybazowany
*)
METHOD PUBLIC HomingGetDone : BOOL
VAR_INPUT
END_VAR
END_METHOD

(*			
	EVERDE sp. z o.o.
	Rafał Osajda		11.04.2025		TC 4024.66
	Zwraca czy bazowanie jest potrzebne
*)
METHOD PUBLIC HomingGetIsNeeded : BOOL
VAR_INPUT
END_VAR
END_METHOD

(*			
	EVERDE sp. z o.o.
	Rafał Osajda		27.05.2025		TC 4024.66
	Uruchomienie metody bazowania
*)
METHOD PUBLIC HomingStart
VAR_INPUT
END_VAR
END_METHOD

(*			
	EVERDE sp. z o.o.
	Rafał Osajda		30.04.2025		TC 4024.66
	Zwraca czy element jest czymś zajety
*)
METHOD PUBLIC IsDoNothing : BOOL
END_METHOD

(*			
	EVERDE sp. z o.o.
	Rafał Osajda		30.04.2025		TC 4024.66
	Zwraca czy element jest w pozycji 0 - referencyjnej
*)
METHOD PUBLIC IsPosition0 : BOOL
END_METHOD

METHOD PUBLIC LinkSS1 : BOOL
VAR_INPUT
	fbSS1			: ITF_BaseFlagGet;
END_VAR
END_METHOD

METHOD PUBLIC LinkSTO : BOOL
VAR_INPUT
	fbSTO			: ITF_BaseFlagGet;
END_VAR
END_METHOD

(*			
	EVERDE sp. z o.o.
	Rafał Osajda		31.03.2025		TC 4024.66
	Zwraca status zasilania	
*)
METHOD PUBLIC PowerGetStatus : BOOL
VAR_INPUT
END_VAR
END_METHOD

(*			
	EVERDE sp. z o.o.
	Rafał Osajda		31.03.2025		TC 4024.66
	Wyłączenie zasilania
*)
METHOD PUBLIC PowerTurnOff : BOOL
VAR_INPUT
END_VAR
END_METHOD

(*			
	EVERDE sp. z o.o.
	Rafał Osajda		31.03.2025		TC 4024.66
	Uruchomienie zasialania
*)
METHOD PUBLIC PowerTurnOn
VAR_INPUT
END_VAR
END_METHOD

END_INTERFACE

// ---- POUs/A06_FB_BaseGroupElement/ITF_BaseGroupElement.TcIO
INTERFACE ITF_BaseGroupElement EXTENDS ITF_BaseControlElement

METHOD PUBLIC LinkCommunicator : BOOL
VAR_INPUT
	fbCommunicator				: ITF_BaseCommunicator;
END_VAR
END_METHOD

END_INTERFACE

// ---- POUs/A06_FB_BaseGroupElement/ITF_BaseGroupElement_HMI_Connector.TcIO
INTERFACE ITF_BaseGroupElement_HMI_Connector EXTENDS ITF_BaseControlElement_HMI_Connector

END_INTERFACE

// ---- POUs/A07_FB_BaseTopElement/ITF_BaseTopElement.TcIO
INTERFACE ITF_BaseTopElement EXTENDS ITF_BaseGroupElement, ITF_BaseSaMStateMethod

METHOD PUBLIC LinkSaM : BOOL
VAR_INPUT
	fbSAM				: ITF_BaseSAM;
END_VAR
END_METHOD

END_INTERFACE

// ---- POUs/A07_FB_BaseTopElement/ITF_BaseTopElement_HMI_Connector.TcIO
INTERFACE ITF_BaseTopElement_HMI_Connector EXTENDS ITF_BaseGroupElement_HMI_Connector

END_INTERFACE

// ---- POUs/B02_Recipes/ITF_BaseCreateTemplateOfRecipe.TcIO
(*			
	RafalOS
	Rafał Osajda		25.10.2025		TC 4024.66
	Dodawanie meteody dla tworzenia szablownow 
*)
INTERFACE ITF_BaseCreateTemplateOfRecipe

METHOD CreateTamplateOfRecipe : BOOL
VAR_INPUT
	itfRecipe				: ITF_BaseCreatingTemplateMethod;	//interfejs do obsługi receptur
END_VAR
END_METHOD

END_INTERFACE

// ---- POUs/B02_Recipes/ITF_BaseCreatingTemplateMethod.TcIO
INTERFACE ITF_BaseCreatingTemplateMethod

(*			
	RafalOS
	Rafał Osajda		25.10.2025		TC 4024.66
	Dodawanie składnika do szablonu
*)
METHOD PUBLIC AddIngredientToTemplate : BOOL
VAR_INPUT
	uiNumber		: UINT;
	stIngredient	: ST_BaseDescriptor;
END_VAR
END_METHOD

(*			
	RafalOS
	Rafał Osajda		25.10.2025		TC 4024.66
	Dodawanie szablonu - metoda wykorzystywana w zewnętrznym FB tworzenia receptur
*)
METHOD PUBLIC AddTemplate : BOOL
VAR_INPUT
	stTexts			: ST_BaseLabel;
END_VAR
END_METHOD

METHOD PUBLIC GetNumberIngredientOFTemplate : UINT
VAR_INPUT
	uiNumber				: UINT;
END_VAR
END_METHOD

METHOD PUBLIC GetNumberOfTemplate : UINT
VAR_INPUT
END_VAR
END_METHOD

END_INTERFACE

// ---- FUNs/CreateElementCode.TcPOU
(*			EVERDE sp. z o.o.
	Rafał Osajda		16.10.2024		TC 4026.11		wer. 0.0.0.1
	Utworzenie kodu elementu 
*)
FUNCTION CreateElementCode : STRING
VAR_INPUT
	sParentCode					: STRING;
	sAdd						: STRING;
END_VAR
VAR
	arrSegments					: ARRAY [0..GVL_BaseConstans.MAX_NESTING_LEVEL] OF STRING;
	iI							: INT;
	iDotPosition				: INT;
	sCodeResult					: STRING;
END_VAR

IF (LEN (STR := sParentCode) > 0) THEN
	arrSegments [0]				:= sParentCode;
	FOR iI := 1 TO TO_INT (GVL_BaseConstans.MAX_NESTING_LEVEL) DO
		iDotPosition			:= find (STR1 := arrSegments [0], STR2 := '.');
		IF (iDotPosition = 0) THEN
			arrSegments [iI]	:= arrSegments [0];
			EXIT;
		ELSE
			arrSegments [iI]	:= LEFT (STR := arrSegments [0], SIZE := iDotPosition - 1);
			arrSegments [0]		:= delete (STR := arrSegments [0], POS := 1, LEN := iDotPosition);
		END_IF
	END_FOR
END_IF
FOR iI := 1 TO TO_INT (GVL_BaseConstans.MAX_NESTING_LEVEL) DO
	IF (arrSegments [iI] = '0' OR arrSegments [iI] = '') THEN
		arrSegments [iI] := sAdd;
		sAdd			:= '0';
	END_IF
	sCodeResult			:= CONCAT (STR1 := sCodeResult, STR2 := arrSegments [iI]);
	IF (iI < TO_INT (GVL_BaseConstans.MAX_NESTING_LEVEL)) THEN
		sCodeResult		:= CONCAT (STR1 := sCodeResult, STR2 := '.');
	END_IF
END_FOR

CreateElementCode							:= sCodeResult;

END_FUNCTION

// ---- POUs Compilation/PRG_Compilation.TcPOU
PROGRAM PRG_Compilation
VAR
	fbLabel					: FB_BaseLabel;
	fbDescription			: FB_BaseDescriptor;
	fbLocation				: FB_BaseLocation;
	fbCommand				: FB_BaseCommand;
	fbImpuls				: FB_BaseImpulse;
	
	sttmpCommonData			: ST_BaseCommonData;

	fbBaseTime				: FB_BaseTime;
	fbBaseCommand			: FB_BaseCommand;
	fbBaseDescriptor		: FB_BaseDescriptor;
	fbBaseFlag				: FB_BaseFlag;
	fbBaseImplulse			: FB_BaseImpulse;
	fbBaseLocation			: FB_BaseLocation;
	
	fbBaseLogger			: FB_BaseLogger;
	fbBaseLoggerElement		: FB_BaseLoggerElement;
	fbBaseComponent			: FB_BaseComponent;
	fbBaseExecutiveElement	: FB_BaseControlElement;
	fbBaseComplexElement	: FB_BaseGroupElement;
	fbBaseMainComponent		: FB_BaseTopElement;
//B
	fbKomunikator		: FB_Communicator;
	fbReceptury			: FB_Recipe;	
END_VAR

END_PROGRAM

// ---- POUs/A00_Basic/FB_BaseLabel.TcPOU
(*			
	RAFALOS
	Rafał Osajda		19.09.2025		TC 4024.66
	
*)
FUNCTION_BLOCK FB_BaseLabel
VAR
	stTexts						: ST_Label;
END_VAR

METHOD PUBLIC GetText : WSTRING
VAR_INPUT
	eLocation				: E_Location;
END_VAR
GetText				:= THIS^.stTexts.arrText [eLocation];
END_METHOD

METHOD PUBLIC GetTexts : ST_Label
VAR_INPUT
END_VAR
GetTexts				:=THIS^.stTexts;
END_METHOD

METHOD PUBLIC SetText
VAR_INPUT
	eLocation			: E_Location;
	wsDescription		: WSTRING;
END_VAR
THIS^.stTexts.arrText [eLocation]	:= wsDescription;
END_METHOD

METHOD PUBLIC SetTexts
VAR_INPUT
	stTexts				: ST_Label;
END_VAR
THIS^.stTexts			:= stTexts;
END_METHOD

END_FUNCTION_BLOCK

// ---- POUs/A00_Basic/FB_BaseDescriptor.TcPOU
(*			
	RAFALOS
	Rafał Osajda		19.09.2025		TC 4024.66
	
*)
FUNCTION_BLOCK FB_BaseDescriptor IMPLEMENTS ITF_BaseDescriptor
VAR
	stDeskryptor					: ST_BaseDescriptor;
END_VAR

METHOD PUBLIC GetDefaultValue : REAL
VAR_INPUT
END_VAR
GetDefaultValue			:= THIS^.stDeskryptor.rDefaultValue;
END_METHOD

METHOD PUBLIC GetDefaultValueFrom : REAL
VAR_INPUT
	stIN				: ST_BaseDescriptor;
END_VAR
GetDefaultValueFrom			:= stIN.rDefaultValue;
END_METHOD

METHOD PUBLIC GetMax : REAL
VAR_INPUT
END_VAR
GetMax					:= THIS^.stDeskryptor.rMax;
END_METHOD

METHOD PUBLIC GetMaxFrom : REAL
VAR_INPUT
	stIN				: ST_BaseDescriptor;
END_VAR
GetMaxFrom				:= stIN.rMax;
END_METHOD

METHOD PUBLIC GetMin : REAL
VAR_INPUT
END_VAR
GetMin				:= THIS^.stDeskryptor.rMin;
END_METHOD

METHOD PUBLIC GetMinFrom : REAL
VAR_INPUT
	stIN			: ST_BaseDescriptor;
END_VAR
GetMinFrom			:= stIN.rMin;
END_METHOD

METHOD PUBLIC GetTexts : ST_BaseLabel
VAR_INPUT
END_VAR
GetTexts				:=THIS^.stDeskryptor.stTexts;
END_METHOD

METHOD PUBLIC GetTextsFrom : ST_BaseLabel
VAR_INPUT
	stIN				: ST_BaseDescriptor;
END_VAR
GetTextsFrom			:=stIN.stTexts;
END_METHOD

METHOD PUBLIC GetUnit : STRING(6)
VAR_INPUT
END_VAR
GetUnit			:= THIS^.stDeskryptor.sUnit;
END_METHOD

METHOD PUBLIC GetUnitFrom : STRING(6)
VAR_INPUT
	stIN			: ST_BaseDescriptor;
END_VAR
GetUnitFrom			:= stIN.sUnit;
END_METHOD

METHOD PUBLIC GetValue : REAL
VAR_INPUT
END_VAR
GetValue			:= this^.stDeskryptor.rValue;
END_METHOD

METHOD PUBLIC GetValueFrom : REAL
VAR_INPUT
	stIN			: ST_BaseDescriptor;
END_VAR
GetValueFrom		:= stIN.rValue;
END_METHOD

METHOD PUBLIC SetDefaultValue
VAR_INPUT
	rDefaultValue: REAL;
END_VAR
THIS^.stDeskryptor.rDefaultValue		:= rDefaultValue;
END_METHOD

METHOD PUBLIC SetDefaultValueIn
VAR_INPUT
	stIN			: REFERENCE TO ST_BaseDescriptor;
	rDefaultValue	: REAL;
END_VAR
stIN.rDefaultValue		:= rDefaultValue;
END_METHOD

METHOD PUBLIC SetMax
VAR_INPUT
	rMax: REAL;
END_VAR
THIS^.stDeskryptor.rMax		:= rMax;
END_METHOD

METHOD PUBLIC SetMaxIn
VAR_INPUT
	stIN			: REFERENCE TO ST_BaseDescriptor;
	rMax: REAL;
END_VAR
stIN.rMax		:= rMax;
END_METHOD

METHOD PUBLIC SetMin
VAR_INPUT
	rMin: REAL;
END_VAR
THIS^.stDeskryptor.rMin		:= rMin;
END_METHOD

METHOD PUBLIC SetMinIn
VAR_INPUT
	stIN			: REFERENCE TO ST_BaseDescriptor;
	rMin: REAL;
END_VAR
stIn.rMin		:= rMin;
END_METHOD

METHOD PUBLIC SetText
VAR_INPUT
	eLocation			: E_BaseLocation;
	wsDescription		: WSTRING;
END_VAR
THIS^.stDeskryptor.stTexts.arrText [eLocation]	:= wsDescription;
END_METHOD

METHOD PUBLIC SetTextIn
VAR_INPUT
	stIN				: REFERENCE TO ST_BaseDescriptor;
	eLocation			: E_BaseLocation;
	wsDescription		: WSTRING;
END_VAR
stIN.stTexts.arrText [eLocation]	:= wsDescription;
END_METHOD

METHOD PUBLIC SetTexts
VAR_INPUT
	stTexts				: ST_BaseLabel;
END_VAR
THIS^.stDeskryptor.stTexts			:= stTexts;
END_METHOD

METHOD PUBLIC SetTextsIn
VAR_INPUT
	stIN				: REFERENCE TO ST_BaseDescriptor;
	stTexts				: ST_BaseLabel;
END_VAR
stIN.stTexts			:= stTexts;
END_METHOD

METHOD PUBLIC SetUnit
VAR_INPUT
	sUnit: STRING(6);
END_VAR
THIS^.stDeskryptor.sUnit		:= sUnit;
END_METHOD

METHOD PUBLIC SetUnitIn
VAR_INPUT
	stIN			: REFERENCE TO ST_BaseDescriptor;
	sUnit: STRING(6);
END_VAR
stIN.sUnit		:= sUnit;
END_METHOD

METHOD PUBLIC SetValue
VAR_INPUT
	rValue: REAL;
END_VAR
THIS^.stDeskryptor.rValue		:= rValue;
END_METHOD

METHOD PUBLIC SetValueIn
VAR_INPUT
	stIN			: REFERENCE TO ST_BaseDescriptor;
	rValue			: REAL;
END_VAR
stIN.rValue			:= rValue;
END_METHOD

END_FUNCTION_BLOCK

// ---- POUs/A00_Basic/FB_BaseLocation.TcPOU
(*			
	RAFALOS
	Rafał Osajda		19.09.2025		TC 4024.66
	Sterowanie językiem systemu
*)
FUNCTION_BLOCK FB_BaseLocation IMPLEMENTS ITF_BaseLocation
VAR
	eLocation		: E_BaseLocation;
	arrLocation		: ARRAY [1..GVL_BaseConstans.NUMBER_OF_LOCATIONS] OF ST_BaseLocationDesctription := 
						[(wsDescription := "Polski", sCode := 'pl'),
						(wsDescription := "English", sCode := 'en'),
						(wsDescription := "German", sCode := 'de')];;
END_VAR

(*			
	RAFALOS
	Rafał Osajda		24.09.2025		TC 4024.66
	Zwraca kod jezyka tzn 
*)
METHOD PUBLIC GetActualCode : STRING
VAR_INPUT
END_VAR
GetActualCode				:= THIS^.arrLocation [THIS^.eLocation].sCode;
END_METHOD

METHOD PUBLIC GetActualDescription : WSTRING
VAR_INPUT
END_VAR
GetActualDescription			:= THIS^.arrLocation [THIS^.eLocation].wsDescription;
END_METHOD

METHOD PUBLIC GetCode : STRING(5)
VAR_INPUT
	iIN				: INT;
END_VAR
GetCode					:= THIS^.arrLocation [iIN].sCode;
END_METHOD

METHOD PUBLIC GetDescription : WSTRING
VAR_INPUT
	iIN				: INT;
END_VAR
GetDescription				:= THIS^.arrLocation [iIN].wsDescription;
END_METHOD

METHOD PUBLIC GetLocation : E_BaseLocation
VAR_INPUT
END_VAR
GetLocation			:= THIS^.eLocation;
END_METHOD

METHOD PUBLIC SetLocation : BOOL
VAR_INPUT
	sLocation				: STRING;
END_VAR
IF (sLocation = TO_STRING (E_BaseLocation.pl)) THEN
	THIS^.eLocation		:= E_BaseLocation.pl;
	SetLocation			:= TRUE;
ELSIF (sLocation = TO_STRING (E_BaseLocation.en)) THEN
	THIS^.eLocation		:= E_BaseLocation.en;
	SetLocation			:= TRUE;
ELSIF (sLocation = TO_STRING (E_BaseLocation.de)) THEN
	THIS^.eLocation		:= E_BaseLocation.de;
	SetLocation			:= TRUE;
END_IF
END_METHOD

END_FUNCTION_BLOCK

// ---- POUs/A00_Basic/FB_BaseCommand.TcPOU
(*			
	RAFALOS
	Rafał Osajda		19.09.2025		TC 4024.66
	
*)
FUNCTION_BLOCK FB_BaseCommand
VAR
	bStatus								: BOOL	:= TRUE;	//flaga informująca o tym czy polecenia aktywne czy nie  - DONE
	bFirstCycle							: BOOL;
	bLastCycle							: BOOL;
	bExecute							: BOOL;				//wlączanie polecenia
	bBusy								: BOOL;				//trwa - BUSY
	bDone								: BOOL	:= TRUE;	// informacja że polecenie zakończyło sie pomyślnie
	iExternalCommandMethodStep			: INT	:= 0;		//krok używany w metodzie zewnętrzej polecenia poprzez dostepne metody
	iInternalCommandMethodStep			: INT 	:= 0;		//Krok Wywoływania Metody Polecenia - krok 
	bAborted							: BOOL;
END_VAR

(*			
	RafalOS
	Rafał Osajda		04.11.2025		TC 4024.66
	Przerwanie pracy polecenia i wyzerowanie zmiennych wystawienie zmiennej Abort
*)
METHOD PUBLIC Abort
VAR_INPUT
END_VAR
THIS^.bStatus							:= TRUE;
THIS^.bExecute							:= FALSE;
THIS^.bBusy								:= FALSE;
THIS^.bDone								:= FALSE;
THIS^.iExternalCommandMethodStep		:= 0;
THIS^.iInternalCommandMethodStep		:= 0;
THIS^.bFirstCycle						:= FALSE;
THIS^.bLastCycle						:= FALSE;
THIS^.bAborted							:= TRUE;
END_METHOD

(*			
	RafalOS
	Rafał Osajda		04.11.2025		TC 4024.66
	Uruchomienie polecenia
*)
METHOD PUBLIC Execute
VAR_INPUT
	
END_VAR
THIS^.bExecute			:= TRUE;
END_METHOD

METHOD PUBLIC GetStep : INT
VAR_INPUT
END_VAR
GetStep				:= THIS^.iExternalCommandMethodStep;
END_METHOD

(*			
	RafalOS
	Rafał Osajda		04.11.2025		TC 4024.66
	Zwraca czy rozkaz został przerwany
*)
METHOD PUBLIC IsAborted : BOOL
VAR_INPUT
END_VAR
IsAborted			:= THIS^.bAborted;
END_METHOD

(*			
	RafalOS
	Rafał Osajda		04.11.2025		TC 4024.66
	Zwraca czy rozkaz jest w trakcie pracy
*)
METHOD PUBLIC IsBusy : BOOL
VAR_INPUT
END_VAR
IsBusy			:= THIS^.bBusy;
END_METHOD

(*			
	RafalOS
	Rafał Osajda		04.11.2025		TC 4024.66
	Zwraca czy rozkas się wykonał
*)
METHOD PUBLIC IsDone : BOOL
VAR_INPUT
END_VAR
IsDone		:= THIS^.bDone;
END_METHOD

METHOD PUBLIC IsFirstCycle : BOOL
VAR_INPUT
END_VAR
IsFirstCycle				:= THIS^.bFirstCycle;
END_METHOD

METHOD PUBLIC IsLastCycle : BOOL
VAR_INPUT
END_VAR
IsLastCycle				:= THIS^.bLastCycle;
END_METHOD

METHOD PUBLIC IsStatus : BOOL
VAR_INPUT
END_VAR
IsStatus		:= THIS^.bStatus;
END_METHOD

(*			
	RafalOS
	Rafał Osajda		03.05.2025		TC 4024.66
	Metoda wykonywana co cykl - jako wejście przyjmuje czy cykl polecenia się skończył czy nie - jak false czyli się skończył to ustawia flagę ostatniego cyklu
*)
METHOD Operation : BOOL
VAR_INPUT
	bIN			: BOOL;
END_VAR
IF (NOT bIN) THEN
	THIS^.bLastCycle						:= TRUE;
END_IF
END_METHOD

(*			
	RafalOS
	Rafał Osajda		03.05.2025		TC 4024.66
	Metoda wykonywana co cykl sprawdza czy jest uruchomone polecenie 
*)
METHOD OperationExecute : BOOL
CASE THIS^.iInternalCommandMethodStep OF
0	:
	IF (THIS^.bBusy AND NOT THIS^.bFirstCycle) THEN
		THIS^.bFirstCycle					:= TRUE;
		THIS^.iInternalCommandMethodStep	:= 10;
		OperationExecute					:= FALSE;
	END_IF
10	:
	THIS^.bFirstCycle						:= FALSE;
	IF (THIS^.bLastCycle) THEN
		THIS^.bLastCycle					:= FALSE;
		THIS^.iInternalCommandMethodStep	:= 0;
		THIS^.bBusy							:= FALSE;
		THIS^.bDone							:= TRUE;
		THIS^.bStatus						:= TRUE;
		OperationExecute					:= FALSE;
	ELSE
		OperationExecute					:= TRUE;
	END_IF
END_CASE
END_METHOD

METHOD PUBLIC Reset
THIS^.bStatus							:= TRUE;
THIS^.bExecute							:= FALSE;
THIS^.bBusy								:= FALSE;
THIS^.bDone								:= FALSE;
THIS^.iExternalCommandMethodStep		:= 0;
THIS^.iInternalCommandMethodStep		:= 0;
THIS^.bFirstCycle						:= FALSE;
THIS^.bLastCycle						:= FALSE;
THIS^.bAborted							:= FALSE;
END_METHOD

(*			
	RAFALOS
	Rafał Osajda		24.09.2025		TC 4024.66
	ustawoienie kroku zewnętrznej metody
*)
METHOD PUBLIC SetStep
VAR_INPUT
	iIn				: int;
END_VAR
THIS^.iExternalCommandMethodStep			:= iIn;
END_METHOD

METHOD PUBLIC SetStepAsFinal : BOOL
VAR_INPUT
END_VAR
THIS^.iExternalCommandMethodStep			:= GVL_BaseConstans.FINISH_STEP;
END_METHOD

METHOD PUBLIC SetStepINC1 : BOOL
VAR_INPUT
END_VAR
THIS^.iExternalCommandMethodStep			:= THIS^.iExternalCommandMethodStep + 1;
END_METHOD

METHOD PUBLIC SetStepINC10 : BOOL
VAR_INPUT
END_VAR
THIS^.iExternalCommandMethodStep			:= THIS^.iExternalCommandMethodStep + 10;
END_METHOD

METHOD PUBLIC SetStepINC5 : BOOL
VAR_INPUT
END_VAR
THIS^.iExternalCommandMethodStep			:= THIS^.iExternalCommandMethodStep + 5;
END_METHOD

(*			
	RafalOS
	Rafał Osajda		03.05.2025		TC 4024.66
	Metoda wykonywana co cykl testująca czy ma się polecenie wykonać
*)
METHOD PUBLIC Test : BOOL
VAR_INPUT
END_VAR
IF (THIS^.bExecute AND NOT THIS^.bBusy) THEN
	THIS^.iExternalCommandMethodStep	:= 0;
	THIS^.bStatus						:= FALSE;
	THIS^.bDone							:= FALSE;
	THIS^.bBusy							:= TRUE;
	THIS^.bExecute						:= FALSE;
	THIS^.bLastCycle					:= FALSE;
	THIS^.bFirstCycle					:= FALSE;	//zmienione z true przy reogranizacji 
	THIS^.iInternalCommandMethodStep	:= 0;
	THIS^.bAborted						:= FALSE;
	Test								:= TRUE;
	
END_IF
END_METHOD

METHOD PUBLIC TestingLastCycle : BOOL
VAR_INPUT
END_VAR
IF (THIS^.iExternalCommandMethodStep = GVL_BaseConstans.FINISH_STEP) THEN
	TestingLastCycle					:= FALSE;
ELSE
	TestingLastCycle					:= TRUE;
END_IF
END_METHOD

(*			
	RafalOS
	Rafał Osajda		03.05.2025		TC 4024.66
	Metoda wylacza zgloszone uruchomienie
*)
METHOD PUBLIC TurnOff : BOOL
VAR_INPUT
END_VAR
THIS^.bExecute		:= FALSE;
END_METHOD

END_FUNCTION_BLOCK

// ---- POUs/A00_Basic/FB_BaseImpulse.TcPOU
FUNCTION_BLOCK FB_BaseImpulse IMPLEMENTS ITF_BaseImpulse
VAR
	tExitOn				: TON;
	tExitOff			: TON;
	rExitOn				: REAL;
	rExitOff			: REAL;
	
	bExecute			: BOOL;
	bFlashing			: BOOL;
	bExit				: BOOL;
	
END_VAR

THIS^.tExitOn 	(IN := (NOT THIS^.tExitOff.Q AND THIS^.bExecute AND THIS^.bFlashing),PT := REAL_TO_TIME (THIS^.rExitOn));
THIS^.tExitOff 	(IN := (THIS^.tExitOn.Q),PT := REAL_TO_TIME (THIS^.rExitOff));

THIS^.bExit		:= (NOT THIS^.tExitOn.Q AND THIS^.bFlashing) OR (THIS^.bExecute AND NOT THIS^.bFlashing);

METHOD PUBLIC GetExit : BOOL
VAR_INPUT
END_VAR
GetExit				:= THIS^.bExit;
END_METHOD

METHOD PUBLIC Reset : BOOL
VAR_INPUT
END_VAR
THIS^.bExecute			:= FALSE;
THIS^.bFlashing			:= FALSE;
THIS^.bExit				:= FALSE;

Reset					:= TRUE;
END_METHOD

METHOD PUBLIC SetExecuteOff
VAR_INPUT
END_VAR
THIS^.bExecute				:= FALSE;
THIS^.bFlashing				:= FALSE;
END_METHOD

METHOD PUBLIC SetExecuteOn
VAR_INPUT
END_VAR
THIS^.bExecute			:= TRUE;
END_METHOD

METHOD PUBLIC SetFlashing
VAR_INPUT
	bIN				: BOOL;
END_VAR
THIS^.bFlashing				:= bIN;
END_METHOD

METHOD PUBLIC SetTimeOff
VAR_INPUT
	rIN: REAL;
END_VAR
THIS^.rExitOff			:= rIN;
END_METHOD

METHOD PUBLIC SetTimeOn
VAR_INPUT
	rIN					: REAL;
END_VAR
THIS^.rExitOn			:= rIN;
END_METHOD

END_FUNCTION_BLOCK

// ---- POUs/A00_Basic/FB_BaseTime.TcPOU
(*			
	RAFALOS
	Rafał Osajda		19.09.2025		TC 4024.66
	Obsługa czasu w systemie
*)
FUNCTION_BLOCK FB_BaseTime IMPLEMENTS ITF_BaseTime
VAR
	fbLokalTime								: Tc2_Utilities.FB_LocalSystemTime;	//pobieranie czasu
	stActualTime							: Tc2_Utilities.TIMESTRUCT;			//przychowywanie czasu
END_VAR

(*			
	RafalOS
	Rafał Osajda		01.09.2025		TC 4024.66
	Konwetrtuje DT to string do postaci DD/MM/YYYY GG:MM:SS
*)
METHOD PUBLIC BaseDTToString : STRING
VAR_INPUT
	inDT					: DT;
END_VAR
VAR
    stTime 					: Tc2_Utilities.TIMESTRUCT;
    sYear, sMonth, sDay 	: STRING(4);
    sHour, sMin, sSec 		: STRING(2);
END_VAR
// Rozbijamy DT na strukturę
stTime := DT_TO_SYSTEMTIME (inDT);

// Konwersja na stringi z zerami wiodącymi
sYear  := UDINT_TO_STRING(stTime.wYear);

sMonth := RIGHT(CONCAT('0', UINT_TO_STRING(stTime.wMonth)), 2);
sDay   := RIGHT(CONCAT('0', UINT_TO_STRING(stTime.wDay)), 2);
sHour  := RIGHT(CONCAT('0', UINT_TO_STRING(stTime.wHour)), 2);
sMin   := RIGHT(CONCAT('0', UINT_TO_STRING(stTime.wMinute)), 2);
sSec   := RIGHT(CONCAT('0', UINT_TO_STRING(stTime.wSecond)), 2);

// Format końcowy: DD/MM/YYYY HH:MM:SS
BaseDTToString := CONCAT(
                CONCAT(CONCAT(sDay, '/'), CONCAT(sMonth, '/')),
                CONCAT(CONCAT(sYear, ' '), 
                    CONCAT(CONCAT(sHour, ':'), 
                        CONCAT(CONCAT(sMin, ':'), sSec)
                    )
                )
             );
END_METHOD

(*			
	RafalOS
	Rafał Osajda		01.09.2025		TC 4024.66
	Konwetrtuje DT to string do postaci DD_MM_YYYY GG_MM_SS - wersja do nazywania plików logów
*)
METHOD PUBLIC BaseDTToString_ : STRING
VAR_INPUT
	inDT				: DT;
END_VAR
VAR
    stTime 					: Tc2_Utilities.TIMESTRUCT;
    sYear, sMonth, sDay 	: STRING(4);
    sHour, sMin, sSec 		: STRING(2);
END_VAR
// Rozbijamy DT na strukturę
stTime := DT_TO_SYSTEMTIME (inDT);

// Konwersja na stringi z zerami wiodącymi
sYear  := UDINT_TO_STRING(stTime.wYear);
sMonth := CONCAT(SEL(stTime.wMonth < 10, '', '0'), UDINT_TO_STRING(stTime.wmonth));
sDay   := CONCAT(SEL(stTime.wday   < 10, '', '0'), UDINT_TO_STRING(stTime.wday));
sHour  := CONCAT(SEL(stTime.whour  < 10, '', '0'), UDINT_TO_STRING(stTime.whour));
sMin   := CONCAT(SEL(stTime.wminute< 10, '', '0'), UDINT_TO_STRING(stTime.wminute));
sSec   := CONCAT(SEL(stTime.wsecond< 10, '', '0'), UDINT_TO_STRING(stTime.wsecond));

// Format końcowy: YYYY-MM-DD_HH-MM-SS
BaseDTToString_ := CONCAT(
                        CONCAT(CONCAT(sDAY, '-'), CONCAT(sMonth, '-')),
                        CONCAT(CONCAT(sYear, '_'),
                            CONCAT(CONCAT(sHour, '-'),
                                CONCAT(CONCAT(sMin, '-'), sSec)
                            )
                        )
                     );
END_METHOD

(*			
	RafalOS
	Rafał Osajda		01.09.2025		TC 4024.66
	Konwertuje czas LTIME do stringa z możliwością wyłączenia milisekund
*)
METHOD PUBLIC BaseLTimeToString : STRING
VAR_INPUT
	ltTime				: LTIME;
	bShowMS			: BOOL;
END_VAR
VAR
	ulNsTotal 			: ULINT;
    uliMsTotal   	  	: ULINT;

    udiDays      	  	: UDINT;
    udiHours     	  	: UDINT;
    udiMinutes   	  	: UDINT;
    udiSeconds   	  	: UDINT;
    udiMs        	  	: UDINT;
	sResult				: STRING;
END_VAR
ulNsTotal 	:= LTIME_TO_ULINT (ltTime);    // LTIME → ULINT (ns)
uliMsTotal 	:= ulNsTotal / 1000000; // ns → ms


// rozbijamy na jednostki
udiDays    	:= TO_UDINT (uliMsTotal / 86400000);           // dni
udiHours    := TO_UDINT ((uliMsTotal MOD 86400000) / 3600000);
udiMinutes  := TO_UDINT ((uliMsTotal MOD 3600000) / 60000);
udiSeconds  := TO_UDINT ((uliMsTotal MOD 60000) / 1000);
udiMs       := TO_UDINT (uliMsTotal MOD 1000);

// budowanie stringa
sResult := '';

sResult := CONCAT(sResult, THIS^.FormatTwoCharacter (udiValue := udiDays));
sResult := CONCAT(sResult, 'd:');
sResult := CONCAT(sResult, THIS^.FormatTwoCharacter (udiValue := udiHours));
sResult := CONCAT(sResult, ':');
sResult := CONCAT(sResult, THIS^.FormatTwoCharacter (udiValue := udiMinutes));
sResult := CONCAT(sResult, ':');
sResult := CONCAT(sResult, THIS^.FormatTwoCharacter (udiValue := udiSeconds));

IF bShowMS THEN
    sResult := CONCAT(sResult, '.');
    sResult := CONCAT(sResult, THIS^.FormatThreeCharacter (udiValue := udiMs));
END_IF

BaseLTimeToString		:= sResult;
END_METHOD

(*			
	RafalOS
	Rafał Osajda		01.09.2025		TC 4024.66
	Konwertuje czas LTIME do stringa z możliwością wybrnia co ma być pokazywane do postaci DDDd:GG:MM:SS:MS
	dni nie rodziala na miesiące i lata 
*)
METHOD PUBLIC BaseLTimeToString_WhatShow : STRING
VAR_INPUT
	ltTime				: LTIME;
	bSwahDays			: BOOL;
	bShowHours			: BOOL;
	bShowMinutes		: BOOL;
	bShowSeconds		: BOOL;
	bShowMS				: BOOL;
END_VAR
VAR
	ulNsTotal 			: ULINT;
    uliMsTotal   	  	: ULINT;

    udiDays      	  	: UDINT;
    udiHours     	  	: UDINT;
    udiMinutes   	  	: UDINT;
    udiSeconds   	  	: UDINT;
    udiMs        	  	: UDINT;
	sResult				: STRING;
END_VAR
ulNsTotal 	:= LTIME_TO_ULINT (ltTime);    // LTIME → ULINT (ns)
uliMsTotal 	:= ulNsTotal / 1000000; // ns → ms


// rozbijamy na jednostki
udiDays    	:= TO_UDINT (uliMsTotal / 86400000);           // dni
udiHours    := TO_UDINT ((uliMsTotal MOD 86400000) / 3600000);
udiMinutes  := TO_UDINT ((uliMsTotal MOD 3600000) / 60000);
udiSeconds  := TO_UDINT ((uliMsTotal MOD 60000) / 1000);
udiMs       := TO_UDINT (uliMsTotal MOD 1000);

// budowanie stringa
sResult := '';

IF bSwahDays THEN
	sResult := CONCAT(sResult, THIS^.FormatTwoCharacter (udiValue := udiDays));
	sResult := CONCAT(sResult, 'd:');
END_IF
IF bShowHours THEN
	sResult := CONCAT(sResult, THIS^.FormatTwoCharacter (udiValue := udiHours));
	sResult := CONCAT(sResult, ':');
END_IF
IF bShowMinutes THEN
	sResult := CONCAT(sResult, THIS^.FormatTwoCharacter (udiValue := udiMinutes));
	sResult := CONCAT(sResult, ':');
END_IF
IF bShowSeconds THEN
	sResult := CONCAT(sResult, THIS^.FormatTwoCharacter (udiValue := udiSeconds));
END_IF
IF bShowMS THEN
    sResult := CONCAT(sResult, '.');
    sResult := CONCAT(sResult, THIS^.FormatThreeCharacter (udiValue := udiMs));
END_IF

BaseLTimeToString_WhatShow		:= sResult;
END_METHOD

METHOD PRIVATE FormatThreeCharacter : STRING
VAR_INPUT
    udiValue : ULINT;
END_VAR
IF udiValue < 10 THEN
    FormatThreeCharacter := CONCAT('00', TO_STRING(udiValue));
ELSIF udiValue < 100 THEN
    FormatThreeCharacter := CONCAT('0', TO_STRING(udiValue));
ELSE
    FormatThreeCharacter := TO_STRING(udiValue);
END_IF
END_METHOD

METHOD PRIVATE FormatTwoCharacter : STRING
VAR_INPUT
    udiValue : UDINT;
END_VAR
IF udiValue < 10 THEN
    FormatTwoCharacter := CONCAT('0', TO_STRING(udiValue));
ELSE
    FormatTwoCharacter := TO_STRING(udiValue);
END_IF
END_METHOD

METHOD PUBLIC StampDT : DT
VAR_INPUT
END_VAR
StampDT									:= SYSTEMTIME_TO_DT (TIMESTR := THIS^.stActualTime);
END_METHOD

METHOD PUBLIC Work : BOOL
VAR_INPUT
	bIN				: bool;	//wlacz wyłacz
END_VAR
fbLokalTime(
	sNetID									:= , 
	bEnable									:= bIN, 
	dwCycle									:= 1, 
	dwOpt									:= , 
	tTimeout								:= , 
	bValid									=> Work, 
	systemTime								=> stActualTime, 
	tzID									=> 
);
END_METHOD

END_FUNCTION_BLOCK

// ---- POUs/A00_Basic/FB_BaseFlag.TcPOU
(*			
	RAFALOS
	Rafał Osajda		19.09.2025		TC 4024.66
	
*)
FUNCTION_BLOCK FB_BaseFlag IMPLEMENTS ITF_BaseFlag
VAR
END_VAR

END_FUNCTION_BLOCK

// ---- POUs/A02_FB_BaseLogger/FB_BaseLogger.TcPOU
(*			
	RAFALOS
	Rafał Osajda		19.09.2025		TC 4024.66
	Moduł logujący wszsytkie zgłoszenia
*)
FUNCTION_BLOCK FB_BaseLogger EXTENDS FB_Base IMPLEMENTS ITF_BaseLogger, ITF_BaseLogger_HMI_Connector
VAR
	stBuffer						: ST_BaseEvents_Queue;
	arrItem							: ARRAY  [1..GVL_BaseConstans.MAX_NUMBER_OF_ALL_ITEM] OF ITF_BaseLogger_Item;
	iNumberOfItem					: INT;
	uiNumerOfReportsIntheSystem		: UINT;		//informacja ogólna o ilosc wszystkich zgłoszeń
	bClearMemory					: BOOL;		//czyści pamięć
	bChangeInMemory					: BOOL;		//informacja dla wyświetlania żeby odświerzyć dla ogólnego wyświetlania
	arrInfoForHMI					: ARRAY [0..GVL_BaseConstans.MAX_NUMBER_OF_ALL_ITEM] OF ST_BaseEvents_InformationAboutEventsForHMI;	//ilosc zgloszen dla poszczegolnych elementow
END_VAR
VAR PERSISTENT
	stMemory						: ST_BaseEvents_Memory;			//zapamiętane zgłoszenia
	stNumberOfReports				: ST_BaseEvents_ActiveEvents;	//ilości różnych zgłoszeń
	arrNumberOfReportsForItem		: ARRAY [1..GVL_BaseConstans.MAX_NUMBER_OF_ALL_ITEM] OF ST_BaseEvents_ActiveEvents;
	
END_VAR

	(*	Pobranie z kolejki zgłoszeń i dodanie do pamięci	*)

WHILE THIS^.stBuffer.iNumerOfEvents > 0 DO
	THIS^.BufferFIFOSupport ();
END_WHILE

	(*	Wyczyszczenie pamięci zdarzeń	*)
	
IF (THIS^.bClearMemory) THEN
	THIS^.bClearMemory				:= FALSE;
	Tc2_System.MEMSET (destAddr := ADR (THIS^.stMemory), fillByte := 0, n := SIZEOF (THIS^.stMemory));
	Tc2_System.MEMSET (destAddr := ADR (THIS^.stNumberOfReports), fillByte := 0, n	:= SIZEOF (THIS^.stNumberOfReports));
	Tc2_System.MEMSET (destAddr := ADR (THIS^.arrNumberOfReportsForItem), fillByte := 0, n	:= SIZEOF (THIS^.arrNumberOfReportsForItem));
END_IF

METHOD PUBLIC AddItem : INT
VAR_INPUT
	itfItem				: ITF_BaseLogger_Item;
END_VAR
THIS^.arrItem [itfItem.GetID ()]	:= itfItem;
THIS^.iNumberOfItem					:= THIS^.iNumberOfItem + 1;
AddItem								:= THIS^.iNumberOfItem;
END_METHOD

(*			
	RafalOS
	Rafał Osajda		09.06.2025		TC 4024.66
	Przenisienie danych z kolejki do zgloszen pamiętanych
*)
METHOD PRIVATE BufferFIFOSupport
	(*	W zależnosci od tego czy to jest nowe, aktualizacja czy zokończenie zadanie wykonaj odpowiednie zadanie 	*)

IF (THIS^.stBuffer.iNumerOfEvents > 0) THEN
	CASE THIS^.stBuffer.arrEvents [1].eEventAction OF
		E_BaseEvents_Action.Start		: 	THIS^.BufferFIFOSupportStart ();
		E_BaseEvents_Action.Confirm		: 	THIS^.BufferFIFOSupportConfirm ();
		E_BaseEvents_Action.Stop		: 	THIS^.BufferFIFOSupportStop ();
	END_CASE
	
(*		przesuniecie danych w kolejce o 1 i zmniejszenie liczy w kolejce o jeden 	*)
	
	Tc2_System.MEMCPY (
		destAddr			:= ADR (THIS^.stBuffer.arrEvents [1]),
		srcAddr				:= ADR (THIS^.stBuffer.arrEvents [2]),
		n					:= (SIZEOF (THIS^.stBuffer.arrEvents [1]) * TO_UINT (THIS^.stBuffer.iNumerOfEvents))
	);
	THIS^.stBuffer.iNumerOfEvents	:= THIS^.stBuffer.iNumerOfEvents - 1;
END_IF
END_METHOD

(*			
	RafalOS
	Rafał Osajda		09.06.2025		TC 4024.66
	znalezienie w pamiętach odpowiedniego wiersza i przepisanie danych 
*)
METHOD PRIVATE BufferFIFOSupportConfirm
VAR_INPUT
END_VAR

VAR
	iI: INT;
END_VAR
//szukanie w tablicy pamiętanych danych z pierwszego wierszza kolejki 

FOR iI := 1 TO TO_INT (THIS^.stMemory.iNumberOfRow) DO 
	IF (THIS^.stMemory.arrRow [iI].uiIDEvent = THIS^.stBuffer.arrEvents [1].uiIDEvent AND
    	(THIS^.stMemory.arrRow [iI].bConfirm AND NOT THIS^.stMemory.arrRow [iI].bConfirmed)) THEN
		THIS^.stMemory.arrRow [iI].bConfirmed	:= TRUE;
		THIS^.stMemory.arrRow [iI].dtConfirmed	:= THIS^.stBuffer.arrEvents [1].dtConfirmed;
		THIS^.ReduceTheNumberOfConfirmations ();
		THIS^.ReduceTheNumberOfConfirmationsForItem (uiIDItem := THIS^.stMemory.arrRow [iI].uiIDItem);
		EXIT;
	END_IF
END_FOR
END_METHOD

(*			
	RafalOS
	Rafał Osajda		09.06.2025		TC 4024.66
	Przenisienie pamietanych o jeden, zwiekszenie liczby pamietanych o jeden 
	przekopiowanie z koeljki wiersz 1 
*)
METHOD PRIVATE BufferFIFOSupportStart
VAR_INPUT
END_VAR
	(*	Aktualizacja lości wierszy pamiętanych	*)
IF (THIS^.stMemory.iNumberOfRow + 1 <= TO_INT (GVL_BaseConstans.MAX_EVENTS_IN_MEMORY)) THEN
	THIS^.stMemory.iNumberOfRow			:= THIS^.stMemory.iNumberOfRow + 1;
ELSE
	THIS^.DecreaseTheNumberOfReports (stRow := THIS^.stMemory.arrRow [GVL_BaseConstans.MAX_EVENTS_IN_MEMORY]);
	THIS^.DecreaseTheNumberOfReportsForItem (stRow := THIS^.stMemory.arrRow [GVL_BaseConstans.MAX_EVENTS_IN_MEMORY]);
END_IF
	(*	Przesunięcie danych w pamięci o jeden i wyczyszczenie zawartości wiersza 1	*)
Tc2_System.MEMMOVE (destAddr := ADR (THIS^.stMemory.arrRow [2]), srcAddr := ADR (THIS^.stMemory.arrRow [1]),n := (SIZEOF (THIS^.stMemory.arrRow [1]) * TO_UINT (THIS^.stMemory.iNumberOfRow)));
Tc2_System.MEMSET (destAddr := ADR (THIS^.stMemory.arrRow [1]), fillByte := 0, n := SIZEOF (THIS^.stMemory.arrRow [1]));
	(*	Przepisanie danych	do wiersza pierwszego	*)
THIS^.stmemory.arrRow [1].bActive				:= THIS^.stBuffer.arrEvents [1].bActive;
THIS^.stmemory.arrRow [1].bIgnoreRepetitions	:= THIS^.stBuffer.arrEvents [1].bIgnoreRepetitions;
THIS^.stmemory.arrRow [1].eEventCategory		:= THIS^.stBuffer.arrEvents [1].eEventCategory;
THIS^.stmemory.arrRow [1].uiIDEvent				:= THIS^.stBuffer.arrEvents [1].uiIDEvent;
THIS^.stmemory.arrRow [1].uiRepetitionCounter	:= THIS^.stBuffer.arrEvents [1].uiRepetitionCounter;
THIS^.stmemory.arrRow [1].dtStart				:= THIS^.stBuffer.arrEvents [1].dtStart;
THIS^.stmemory.arrRow [1].bConfirm				:= THIS^.stBuffer.arrEvents [1].bConfirm;
THIS^.stmemory.arrRow [1].uiIDItem				:= THIS^.stBuffer.arrEvents [1].uiIDItem;

THIS^.arrInfoForHMI [THIS^.stBuffer.arrEvents [1].uiIDItem].bNew		:= TRUE;
THIS^.arrInfoForHMI [THIS^.stBuffer.arrEvents [1].uiIDItem].iQuantity	:= THIS^.arrInfoForHMI [THIS^.stBuffer.arrEvents [1].uiIDItem].iQuantity + 1;
THIS^.bChangeInMemory		:= TRUE;
(*	informacja dla systemu że jest aktywny błąd 	*)
THIS^.IncreaseTheNumberOfReports (stRow := THIS^.stMemory.arrRow [1]);
THIS^.IncreaseTheNumberOfReportsForItem (stRow := THIS^.stMemory.arrRow [1]);
END_METHOD

(*			
	RafalOS
	Rafał Osajda		09.06.2025		TC 4024.66
	Znalezienie w pamieci odpowiedniego wiersza i przypisanie odpowiednich danych stempel i zmiena flagi
*)
METHOD PRIVATE BufferFIFOSupportStop
VAR_INPUT
END_VAR

VAR
	iI: INT;
END_VAR
FOR iI := 1 TO TO_INT (THIS^.stMemory.iNumberOfRow) DO 
	IF (THIS^.stMemory.arrRow [iI].uiIDEvent = THIS^.stBuffer.arrEvents [1].uiIDEvent AND
		((THIS^.stMemory.arrRow [iI].bConfirm AND THIS^.stMemory.arrRow [iI].bConfirmed AND
			THIS^.stMemory.arrRow [iI].dtFinish = DT#1970-1-1-0:0:0) OR NOT THIS^.stMemory.arrRow [iI].bConfirm)) THEN
		THIS^.stMemory.arrRow [iI].bActive		:= FALSE;
		THIS^.stMemory.arrRow [iI].dtFinish		:= THIS^.stBuffer.arrEvents [1].dtFinish;
		THIS^.ReduceTheNumberOfActiveEvents (eEventsCategory	:= THIS^.stMemory.arrRow [iI].eEventCategory);
		THIS^.ReduceTheNumberOfActiveEventsForItem (uiIDItem := THIS^.stMemory.arrRow [iI].uiIDItem, eEventsCategory := THIS^.stMemory.arrRow [iI].eEventCategory);
		EXIT;
	END_IF
END_FOR
END_METHOD

METHOD PRIVATE DecreaseTheNumberOfReports
VAR_INPUT
	stRow					: ST_BaseEvents_RowInMemory;
END_VAR
VAR
	bConfirm				: BOOL;
	eEventsCategory			: E_BaseEvents_Category;
END_VAR
bConfirm					:= stRow.bConfirm;
eEventsCategory				:= stRow.eEventCategory;

IF (stRow.bActive) THEN
	THIS^.stNumberOfReports.iNumberOfActive					:= THIS^.stNumberOfReports.iNumberOfActive - 1;
END_IF
THIS^.stNumberOfReports.bIsActive							:= THIS^.stNumberOfReports.bIsActive > 0;
IF (bConfirm) THEN
	THIS^.stNumberOfReports.iNumberOfActiveWithConfirmation	:= THIS^.stNumberOfReports.iNumberOfActiveWithConfirmation - 1;
	THIS^.stNumberOfReports.bIsActiveWithConfirmation		:= THIS^.stNumberOfReports.bIsActiveWithConfirmation > 0;
END_IF

THIS^.stNumberOfReports.arrNumberOfActive [eEventsCategory]	:= THIS^.STNumberOfReports.arrNumberOfActive [eEventsCategory] - 1;
THIS^.stNumberOfReports.iTotalNumer							:= THIS^.stNumberOfReports.iTotalNumer - 1;
THIS^.stNumberOfReports.arrTotalNumer [eEventsCategory]		:= THIS^.stNumberOfReports.arrTotalNumer [eEventsCategory] - 1;
THIS^.stNumberOfReports.arrActive [eEventsCategory]			:= THIS^.stNumberOfReports.arrNumberOfActive [eEventsCategory] > 0;
END_METHOD

METHOD PRIVATE DecreaseTheNumberOfReportsForItem
VAR_INPUT
	stRow					: ST_BaseEvents_RowInMemory;
END_VAR
VAR
	uiIDItem				: UINT;
	bConfirm				: BOOL;
	eEventsCategory			: E_BaseEvents_Category;
END_VAR
uiIDItem					:= stRow.uiIDItem;
bConfirm					:= stRow.bConfirm;
eEventsCategory				:= stRow.eEventCategory;

IF (stRow.bActive) THEN
	THIS^.stNumberOfReports.iNumberOfActive						:= THIS^.stNumberOfReports.iNumberOfActive - 1;
END_IF
THIS^.stNumberOfReports.bIsActive							:= THIS^.stNumberOfReports.bIsActive > 0;
IF (bConfirm) THEN
	THIS^.stNumberOfReports.iNumberOfActiveWithConfirmation	:= THIS^.stNumberOfReports.iNumberOfActiveWithConfirmation - 1;
	THIS^.stNumberOfReports.bIsActiveWithConfirmation		:= THIS^.stNumberOfReports.bIsActiveWithConfirmation > 0;
END_IF

THIS^.stNumberOfReports.arrNumberOfActive [eEventsCategory]	:= THIS^.STNumberOfReports.arrNumberOfActive [eEventsCategory] - 1;
THIS^.stNumberOfReports.iTotalNumer							:= THIS^.stNumberOfReports.iTotalNumer - 1;
THIS^.stNumberOfReports.arrTotalNumer [eEventsCategory]		:= THIS^.stNumberOfReports.arrTotalNumer [eEventsCategory] - 1;
THIS^.stNumberOfReports.arrActive [eEventsCategory]			:= THIS^.stNumberOfReports.arrNumberOfActive [eEventsCategory] > 0;
END_METHOD

(*			
	RafalOS
	Rafał Osajda		02.10.2025		TC 4024.66
	Zwraca czy nastąpiła jakaś zmiana w pamięci zgłoszeń - całej nie tylko dla jakiegoś elementu
*)
METHOD PUBLIC GetChangeInMemory : BOOL
VAR_INPUT
END_VAR
GetChangeInMemory			:= THIS^.bChangeInMemory;
END_METHOD

METHOD PUBLIC GetEventCounts : ST_BaseEvents_ActiveEvents
VAR_INPUT
END_VAR
GetEventCounts			:= THIS^.stNumberOfReports;
END_METHOD

METHOD PUBLIC GetEventCountsForItem : ST_BaseEvents_ActiveEvents
VAR_INPUT
	uiIDItem: UINT;
END_VAR
GetEventCountsForItem		:= THIS^.arrNumberOfReportsForItem [uiIDItem];
END_METHOD

METHOD PUBLIC GetInformationFromItem : ST_BaseLogger_ItemDataToDisplay
VAR_INPUT
	uiIDItem				: UINT;
	uiIDEvent				: UINT;
END_VAR
GetInformationFromItem		:= THIS^.arrItem [uiIDItem].GetInformationToDisplayEvent (uiIDEvent := uiIDEvent);
END_METHOD

METHOD PUBLIC GetNumerOfReportsIntheSystem : UINT
VAR_INPUT
END_VAR
GetNumerOfReportsIntheSystem	:= THIS^.uiNumerOfReportsIntheSystem;
END_METHOD

METHOD GetReferenceToStmemory : REFERENCE TO ST_BaseEvents_Memory
VAR_INPUT
		
END_VAR
GetReferenceToStmemory			REF= THIS^.stMemory;
END_METHOD

METHOD PRIVATE IncreaseTheNumberOfReports
VAR_INPUT
	stRow					: ST_BaseEvents_RowInMemory;
END_VAR
VAR
	bConfirm				: BOOL;
	eEventsCategory			: E_BaseEvents_Category;
END_VAR
bConfirm					:= stRow.bConfirm;
eEventsCategory				:= stRow.eEventCategory;

THIS^.stNumberOfReports.iNumberOfActive						:= THIS^.stNumberOfReports.iNumberOfActive + 1;
THIS^.stNumberOfReports.bIsActive							:= TRUE;
THIS^.stNumberOfReports.iTotalNumer							:= THIS^.stNumberOfReports.iTotalNumer + 1;
IF (bConfirm) THEN
	THIS^.stNumberOfReports.bIsActiveWithConfirmation		:= TRUE;
	THIS^.stNumberOfReports.iNumberOfActiveWithConfirmation	:= THIS^.stNumberOfReports.iNumberOfActiveWithConfirmation + 1;
END_IF

THIS^.stNumberOfReports.arrNumberOfActive [eEventsCategory]	:= THIS^.stNumberOfReports.arrNumberOfActive [eEventsCategory] + 1;
THIS^.stNumberOfReports.arrTotalNumer [eEventsCategory]		:= THIS^.stNumberOfReports.arrTotalNumer [eEventsCategory] + 1;
THIS^.stNumberOfReports.arrActive [eEventsCategory]			:= THIS^.stNumberOfReports.arrNumberOfActive [eEventsCategory] > 0;
END_METHOD

METHOD PRIVATE IncreaseTheNumberOfReportsForItem
VAR_INPUT
	stRow					: ST_BaseEvents_RowInMemory;
END_VAR
VAR
	uiIDItem				: UINT;
	bConfirm				: BOOL;
	eEventsCategory			: E_BaseEvents_Category;
END_VAR
uiIDItem					:= stRow.uiIDItem;
bConfirm					:= stRow.bConfirm;
eEventsCategory				:= stRow.eEventCategory;

THIS^.arrNumberOfReportsForItem [uiIDItem].iNumberOfActive	:= THIS^.arrNumberOfReportsForItem [uiIDItem].iNumberOfActive + 1;
THIS^.arrNumberOfReportsForItem [uiIDItem].bIsActive		:= TRUE;
IF (bConfirm) THEN
	THIS^.arrNumberOfReportsForItem [uiIDItem].bIsActiveWithConfirmation		:= TRUE;
	THIS^.arrNumberOfReportsForItem [uiIDItem].iNumberOfActiveWithConfirmation	:= THIS^.arrNumberOfReportsForItem [uiIDItem].iNumberOfActiveWithConfirmation + 1;
END_IF

THIS^.arrNumberOfReportsForItem [uiIDItem].arrNumberOfActive [eEventsCategory]	:= THIS^.arrNumberOfReportsForItem [uiIDItem].arrNumberOfActive [eEventsCategory] + 1;
THIS^.arrNumberOfReportsForItem [uiIDItem].iTotalNumer							:= THIS^.arrNumberOfReportsForItem [uiIDItem].iTotalNumer + 1;
THIS^.arrNumberOfReportsForItem [uiIDItem].arrTotalNumer [eEventsCategory]		:= THIS^.arrNumberOfReportsForItem [uiIDItem].arrTotalNumer [eEventsCategory] + 1;
THIS^.arrNumberOfReportsForItem [uiIDItem].arrActive [eEventsCategory]			:= THIS^.arrNumberOfReportsForItem [uiIDItem].arrNumberOfActive [eEventsCategory] > 0;
END_METHOD

(*			
	RafalOS
	Rafał Osajda		12.06.2025		TC 4024.66
	Zmniejsza ilosć aktywnych błędów
*)
METHOD PRIVATE ReduceTheNumberOfActiveEvents : BOOL
VAR_INPUT
	eEventsCategory		: E_BaseEvents_Category;
END_VAR
THIS^.stNumberOfReports.iNumberOfActive	:= THIS^.stNumberOfReports.iNumberOfActive - 1;
IF (THIS^.stNumberOfReports.iNumberOfActive = 0) THEN
	THIS^.stNumberOfReports.bIsActive	:= FALSE;
END_IF

THIS^.stNumberOfReports.arrNumberOfActive [eEventsCategory]	:= THIS^.stnumberOfReports.arrNumberOfActive [eEventsCategory] - 1;
THIS^.stNumberOfReports.arrActive [eEventsCategory]			:= THIS^.stnumberOfReports.arrNumberOfActive [eEventsCategory] > 0;
END_METHOD

(*			
	RafalOS
	Rafał Osajda		12.06.2025		TC 4024.66
	Zmniejsza ilosć aktywnych błędów
*)
METHOD PRIVATE ReduceTheNumberOfActiveEventsForItem : BOOL
VAR_INPUT
	uiIDItem			: UINT;
	eEventsCategory		: E_BaseEvents_Category;
END_VAR
THIS^.arrNumberOfReportsForItem [uiIDItem].iNumberOfActive	:= THIS^.arrNumberOfReportsForItem [uiIDItem].iNumberOfActive - 1;
IF (THIS^.arrNumberOfReportsForItem [uiIDItem].iNumberOfActive = 0) THEN
	THIS^.arrNumberOfReportsForItem [uiIDItem].bIsActive	:= FALSE;
END_IF

THIS^.arrNumberOfReportsForItem [uiIDItem].arrNumberOfActive [eEventsCategory]	:= THIS^.arrNumberOfReportsForItem [uiIDItem].arrNumberOfActive [eEventsCategory] - 1;
THIS^.arrNumberOfReportsForItem [uiIDItem].arrActive [eEventsCategory]			:= THIS^.arrNumberOfReportsForItem [uiIDItem].arrNumberOfActive [eEventsCategory] > 0;
END_METHOD

(*			
	RafalOS
	Rafał Osajda		12.06.2025		TC 4024.66
	Zminiejsza ilość potwierdzeń w aktywnych błedach
*)
METHOD PRIVATE ReduceTheNumberOfConfirmations : BOOL
VAR_INPUT
END_VAR
THIS^.stNumberOfReports.iNumberOfActiveWithConfirmation		:= THIS^.stNumberOfReports.iNumberOfActiveWithConfirmation - 1;
IF (THIS^.stNumberOfReports.iNumberOfActiveWithConfirmation = 0) THEN
	THIS^.stNumberOfReports.bIsActiveWithConfirmation	:= FALSE;
END_IF
END_METHOD

(*			
	RafalOS
	Rafał Osajda		12.06.2025		TC 4024.66
	Zminiejsza ilość potwierdzeń w aktywnych błedach
*)
METHOD PRIVATE ReduceTheNumberOfConfirmationsForItem : BOOL
VAR_INPUT
	uiIDItem: UINT;
END_VAR
THIS^.arrNumberOfReportsForItem [uiIDItem].iNumberOfActiveWithConfirmation		:= THIS^.arrNumberOfReportsForItem [uiIDItem].iNumberOfActiveWithConfirmation - 1;
IF (THIS^.arrNumberOfReportsForItem [uiIDItem].iNumberOfActiveWithConfirmation = 0) THEN
	THIS^.arrNumberOfReportsForItem [uiIDItem].bIsActiveWithConfirmation	:= FALSE;
END_IF
END_METHOD

(*			
	RAFALOS
	Rafał Osajda		26.09.2025		TC 4024.66
	Dodanie do kolejki
*)
METHOD PUBLIC ReportEvent : BOOL
VAR_INPUT
	stEvent					: ST_BaseEvents_RowInQueue;
END_VAR
	
	(*		Kolejka FIFO dodajemy na koniec pobieramy z początku	*)
	(*		Dodanie na koniec kolejki	*)
	
IF (THIS^.stBuffer.inumerOfEvents + 1 <= TO_INT (GVL_BaseConstans.MAX_NUMBER_OF_EVENTS_IN_THE_QUEUE)) THEN
	THIS^.stBuffer.iNumerOfEvents								:= THIS^.stBuffer.iNumerOfEvents  + 1;
	THIS^.stBuffer.arrEvents [THIS^.stBuffer.iNumerOfEvents]	:= stEvent;
END_IF
END_METHOD

(*			
	RafalOS
	Rafał Osajda		02.10.2025		TC 4024.66
	
*)
METHOD PUBLIC ResetChangeInMemory : BOOL
VAR_INPUT
END_VAR
THIS^.bChangeInMemory			:= FALSE;
END_METHOD

METHOD PUBLIC SetNumerOfReportsIntheSystem
VAR_INPUT
	uiValue		: UINT;
END_VAR
THIS^.uiNumerOfReportsIntheSystem	:= uiValue;
END_METHOD

END_FUNCTION_BLOCK

// ---- POUs/A01_Base/FB_Base.TcPOU
(*			
	RAFALOS
	Rafał Osajda		22.09.2025		TC 4024.66
	Bazowy FB dla wszystkich elementów systemu, zawiera główne metody dla łaczenia danych
*)
FUNCTION_BLOCK FB_Base EXTENDS FB_BaseDescriptor IMPLEMENTS ITF_Base
VAR
	refstCommonData			: REFERENCE TO ST_BaseCommonData;
	bIsValidCommonData		: BOOL;
END_VAR

METHOD PUBLIC IsValidCommonData : BOOL
VAR_INPUT
END_VAR
IsValidCommonData			:= THIS^.bIsValidCommonData;
END_METHOD

METHOD PUBLIC LinkCommonData : BOOL
VAR_INPUT
	stCommonData				: REFERENCE TO ST_BaseCommonData;
END_VAR
THIS^.refstCommonData			REF= stCommonData;

IF (__ISVALIDREF (THIS^.refstCommonData)) THEN
	THIS^.bIsValidCommonData		:= TRUE;
	LinkCommonData					:= TRUE;
ELSE
	LinkCommonData					:= FALSE;
END_IF
END_METHOD

METHOD PUBLIC SetName
VAR_INPUT
	stName				: ST_BaseLabel;
END_VAR
END_METHOD

END_FUNCTION_BLOCK

// ---- POUs/A03_FB_BaseLoggerElement/FB_BaseLoggerElement.TcPOU
(*			
	RAFALOS
	Rafał Osajda		19.09.2025		TC 4024.66
	Element bazowy umożliwiający potomkom wysyłaś zgłoszenia do logera
*)
FUNCTION_BLOCK FB_BaseLoggerElement EXTENDS FB_Base IMPLEMENTS ITF_BaseLoggerElement, ITF_BaseLoggerElement_HMI_Connector, ITF_BaseLogger_Item, ITF_DecoratedElement
VAR
	stIdentifier					: ST_BaseElementIdentifier;	//Identyfikacja elementu
	stEvents						: ST_BaseEvents;			//dane elementu dotyczące zdarzeń
END_VAR

(*			
	RafalOS
	Rafał Osajda		24.03.2025		TC 4024.66
	Dodawanie zgłoszenia do systemu
*)
METHOD PUBLIC AddEvent : BOOL
VAR_INPUT
	bIgnoreRepetitions					: BOOL;						//jak true nie zliczaj powtorzeń wystapienia np komunikaty
	eEventCategory						: E_BaseEvents_Category;	//BYTE;	//1 - blad, 2 - ostrzezenie, 3 - wiadomosc, 4 - safety
	bConfirm							: BOOL;						//wymaga powtierdzenia
	stDescription						: ST_BaseLabel;
END_VAR
IF (THIS^.stEvents.uiNumberOfAdded + 1 <= GVL_BaseConstans.MAX_EVENTS_PER_ITEM) THEN
	THIS^.stEvents.uiNumberOfAdded														:= THIS^.stEvents.uiNumberOfAdded + 1;
	THIS^.stEvents.arrDefinitions [THIS^.stEvents.uiNumberOfAdded].uiIDInItem			:= THIS^.stEvents.uiNumberOfAdded;
	THIS^.stEvents.arrDefinitions [THIS^.stEvents.uiNumberOfAdded].bIgnoreRepetitions	:= bIgnoreRepetitions;
	THIS^.stEvents.arrDefinitions [THIS^.stEvents.uiNumberOfAdded].eEventCategory		:= eEventCategory;
	THIS^.stEvents.arrDefinitions [THIS^.stEvents.uiNumberOfAdded].stDescription		:= stDescription;
	THIS^.stEvents.arrDefinitions [THIS^.stEvents.uiNumberOfAdded].bConfirm				:= bConfirm;
	AddEvent						:= TRUE;
ELSE
	AddEvent						:= FALSE;
END_IF
END_METHOD

METHOD PROTECTED EventAcknowledge : BOOL
VAR_INPUT
	iNumber				: INT;
END_VAR
VAR
	sttmpRow			: ST_BaseEvents_RowInQueue;
	btmpExit			: BOOL;
END_VAR
IF (iNumber > 0 AND iNumber <= TO_INT (THIS^.stEvents.uiNumberOfAdded)) THEN
	IF ((THIS^.stEvents.arrDefinitions [iNumber].bConfirm AND NOT THIS^.stEvents.arrConfirmation [iNumber]) OR NOT THIS^.stEvents.arrDefinitions [iNumber].bConfirm) THEN
		THIS^.stEvents.arrConfirmation [iNumber] 	:= TRUE;
		btmpExit									:= TRUE;
		IF (THIS^.stEvents.bLoggerDataCompleted) THEN
			sttmpRow.eEventAction		:= E_BaseEvents_Action.Confirm;
			sttmpRow.uiIDEvent			:= THIS^.stEvents.arrDefinitions [iNumber].uiIDEvent;
			sttmpRow.dtConfirmed		:= THIS^.refstCommonData.itfTime.StampDT ();
		
			THIS^.refstCommonData.itfLogger.ReportEvent (stEvent	:= sttmpRow);	
			btmpExit						:= btmpExit;
		ELSE
			btmpExit						:= FALSE;
		END_IF
	END_IF	
END_IF
EventAcknowledge					:= btmpExit;
END_METHOD

(*			
	RafalOS
	Rafał Osajda		09.06.2025		TC 4024.66
	Szuka czy ma zgłoszenie i zadanym ID jak tak to usuwa i zwraca true w przeciwnym razie zwraca false 
*)
METHOD PUBLIC EventAcknowledgeByID : BOOL
VAR_INPUT
	uiIDEvent				: UINT;
END_VAR

VAR
	iI: INT;
	bResult: BOOL;
END_VAR
FOR iI := 1 TO TO_INT (THIS^.stEvents.uiNumberOfAdded) DO
	IF (THIS^.stEvents.arrDefinitions [iI].uiIDEvent = uiIDEvent AND THIS^.stEvents.arrDefinitions [iI].bConfirm) THEN	//Zgłoszenie znalezione
		IF (THIS^.EventAcknowledge (iNumber	:= iI)) THEN
			bResult							:= TRUE;
			EXIT;
		END_IF
	END_IF
END_FOR
EventAcknowledgeByID					:= bResult;
END_METHOD

METHOD PROTECTED EventDoesRequireConfirmation : BOOL
VAR_INPUT
	iNumber				: INT;
END_VAR
EventDoesRequireConfirmation		:= THIS^.stEvents.arrDefinitions [iNumber].bConfirm;
END_METHOD

(*			RafalOS
	Rafał Osajda		16.10.2024		TC 4026.11		wer. 0.0.0.1
	Zwraca aktualny stan wybranego zgłoszenia
*)
METHOD PROTECTED EventIsActive : BOOL
VAR_INPUT
	iNumber					: INT;
END_VAR
IF (iNumber > 0 AND iNumber <= TO_INT (THIS^.stEvents.uiNumberOfAdded)) THEN
	EventIsActive			:= THIS^.stEvents.arrState [iNumber];
END_IF
END_METHOD

(*			
	RafalOS
	Rafał Osajda		24.03.2025		TC 4024.66
	Definicja nowego zgłoszenia
*)
METHOD PUBLIC EventsDefinition : BOOL
MEMSET (
	destAddr		:= ADR (THIS^.stEvents.arrDefinitions),
	fillByte		:= 0,
	n				:= SIZEOF (THIS^.stEvents.arrDefinitions)
);
THIS^.stEvents.uiNumberOfAdded	:= 0;
END_METHOD

(*			
	RafalOS
	Rafał Osajda		24.03.2025		TC 4024.66
	Zgloszenie nowe wlacz 
*)
METHOD PROTECTED EventSetActive : BOOL
VAR_INPUT
	iNumber					: INT; //numer zgloszenia w elemencie
END_VAR
VAR
	sttmpRow				: ST_BaseEvents_RowInQueue;
END_VAR
IF (iNumber > 0 AND iNumber <= TO_INT (THIS^.stEvents.uiNumberOfAdded) AND NOT THIS^.stEvents.arrState [iNumber]) THEN
	THIS^.stEvents.arrState [iNumber]		:= TRUE;
	IF (NOT THIS^.stEvents.arrDefinitions [iNumber].bIgnoreRepetitions) THEN
		THIS^.stEvents.arrDefinitions [iNumber].uiRepetitionCounter := THIS^.stEvents.arrDefinitions [iNumber].uiRepetitionCounter + 1;
	END_IF
	IF (THIS^.stEvents.bLoggerDataCompleted) THEN
		sttmpRow.eEventAction		:= E_BaseEvents_Action.Start;
		sttmpRow.uiIDEvent			:= THIS^.stEvents.arrDefinitions [iNumber].uiIDEvent;
		sttmpRow.bActive			:= TRUE;
		sttmpRow.bIgnoreRepetitions	:= THIS^.stEvents.arrDefinitions [iNumber].bIgnoreRepetitions;
		sttmpRow.dtStart			:= THIS^.refstCommonData.itfTime.StampDT ();
		sttmpRow.uiRepetitionCounter:= THIS^.stEvents.arrDefinitions [iNumber].uiRepetitionCounter;
		sttmpRow.eEventCategory		:= THIS^.stEvents.arrDefinitions [iNumber].eEventCategory;
		sttmpRow.bConfirm			:= THIS^.stEvents.arrDefinitions [iNumber].bConfirm;
		sttmpRow.uiIDItem			:= THIS^.stIdentifier.uiID;
		
		THIS^.refstCommonData.itfLogger.ReportEvent (stEvent := sttmpRow);
		THIS^.stEvents.iNumberOfActiveEvents	:= THIS^.stEvents.iNumberOfActiveEvents + 1;
	END_IF
END_IF
END_METHOD

(*			
	RafalOS
	Rafał Osajda		24.03.2025		TC 4024.66
	Zgloszenie zakonczone wylacz
*)
METHOD PROTECTED EventSetInactive : BOOL
VAR_INPUT
	iNumber				: INT;
END_VAR
VAR
	iI					: INT;
	sttmpRow			: ST_BaseEvents_RowInQueue;
	btmpExit			: BOOL := FALSE;
END_VAR
IF (iNumber > 0 AND iNumber <= TO_INT (THIS^.stEvents.uiNumberOfAdded) AND THIS^.stEvents.arrState [iNumber]) THEN
	IF ((THIS^.stEvents.arrDefinitions [iNumber].bConfirm AND THIS^.stEvents.arrConfirmation [iNumber]) OR NOT THIS^.stEvents.arrDefinitions [iNumber].bConfirm) THEN
		stEvents.arrState [iNumber]					:= FALSE;
		THIS^.stEvents.arrConfirmation [iNumber]	:= FALSE;
		btmpExit									:= TRUE;
	END_IF
	IF (THIS^.stEvents.bLoggerDataCompleted) THEN
		sttmpRow.eEventAction		:= E_BaseEvents_Action.Stop;
		sttmpRow.uiIDEvent			:= THIS^.stEvents.arrDefinitions [iNumber].uiIDEvent;
		sttmpRow.dtFinish			:= THIS^.refstCommonData.itfTime.StampDT ();
		sttmpRow.bActive			:= FALSE;
	
		THIS^.refstCommonData.itfLogger.ReportEvent (stEvent	:= sttmpRow);
		THIS^.stEvents.iNumberOfActiveEvents	:= THIS^.stEvents.iNumberOfActiveEvents - 1;
		btmpExit						:= btmpExit;
	ELSE
		btmpExit						:= FALSE;
	END_IF
END_IF
EventSetInactive 						:= btmpExit;
END_METHOD

(*			
	RafalOS
	Rafał Osajda		09.06.2025		TC 4024.66
	Szuka czy ma zgłoszenie i zadanym ID jak tak to usuwa i zwraca true w przeciwnym razie zwraca false 
*)
METHOD PUBLIC EventSetInactiveByID : BOOL
VAR_INPUT
	uiIDEvent				: UINT;
END_VAR

VAR
	iI: INT;
	bResult: BOOL;
END_VAR
FOR iI := 1 TO TO_INT (THIS^.stEvents.uiNumberOfAdded) DO
	IF (THIS^.stEvents.arrDefinitions [iI].uiIDEvent = uiIDEvent AND
		((NOT THIS^.stEvents.arrDefinitions [iI].bConfirm) OR 
			(THIS^.stEvents.arrDefinitions [iI].bConfirm AND THIS^.stEvents.arrConfirmation [iI]))) THEN	//Zgłoszenie znalezione
		IF (THIS^.EventSetInactive (iNumber := iI)) THEN
			bResult							:= TRUE;
			EXIT;
		END_IF
	END_IF
END_FOR
EventSetInactiveByID						:= bResult;
END_METHOD

(*			
	RAFALOS
	Rafał Osajda		25.09.2025		TC 4024.66
	Metoda wywoływana w pierwszym cyklu
*)
METHOD PUBLIC FirstCycle : BOOL
VAR_INPUT
END_VAR
	(*	Zdefiniowanie zdarzeń dla elementu	*)
THIS^.EventsDefinition ();


FirstCycle					:= TRUE;
END_METHOD

METHOD PUBLIC GetCode : STRING
VAR_INPUT
END_VAR
GetCode			:= THIS^.stIdentifier.sCode;
END_METHOD

METHOD PUBLIC GetID : UINT
VAR_INPUT
END_VAR
GetID				:= THIS^.stIdentifier.uiID;
END_METHOD

METHOD PUBLIC GetIdentyfier : ST_BaseElementIdentifier
VAR_INPUT
END_VAR
GetIdentyfier				:= THIS^.stIdentifier;
END_METHOD

METHOD GetInformationToDisplayEvent : ST_BaseLogger_ItemDataToDisplay
VAR_INPUT
	uiIDEvent				: UINT;
END_VAR
VAR
	sttmpResult				: ST_BaseLogger_ItemDataToDisplay;
	iI: INT;
END_VAR
sttmpResult.stItemName		:= THIS^.stIdentifier.stName;
sttmpResult.sCode			:= THIS^.stIdentifier.sCode;
FOR iI := 1 TO TO_INT (THIS^.stEvents.uiNumberOfAdded) DO 
	IF (THIS^.stEvents.arrDefinitions [iI].uiIDEvent = uiIDEvent) THEN
		sttmpResult.stDescription	:= THIS^.stEvents.arrDefinitions [iI].stDescription;
		sttmpResult.eEventCategory	:= THIS^.stEvents.arrDefinitions [iI].eEventCategory;
		sttmpResult.sEventCategory	:= TO_STRING (THIS^.stEvents.arrDefinitions [iI].eEventCategory);
		sttmpResult.uiRepetitionCounter	:= THIS^.stEvents.arrDefinitions [iI].uiRepetitionCounter;
		EXIT;
	END_IF
END_FOR

GetInformationToDisplayEvent	:= sttmpResult;
END_METHOD

METHOD GetITFComponent : ITF_BaseComponent
VAR_INPUT
END_VAR
GetITFComponent		:= null;
END_METHOD

METHOD GetITFControlElement : ITF_BaseControlElement
VAR_INPUT
END_VAR
GetITFControlElement	:= null;
END_METHOD

METHOD GetITFGroupElement : ITF_BaseGroupElement
VAR_INPUT
END_VAR
GetITFGroupElement	:= null;
END_METHOD

METHOD GetITFLoggerElement : ITF_BaseLoggerElement
VAR_INPUT
END_VAR
GetITFLoggerElement		:= THIS^;
END_METHOD

METHOD GetITFTopElement : ITF_BaseTopElement
VAR_INPUT
END_VAR
GetITFTopElement		:= null;
END_METHOD

METHOD PUBLIC GetName : ST_BaseLabel
VAR_INPUT
END_VAR
GetName				:= THIS^.stIdentifier.stName;
END_METHOD

METHOD PUBLIC GetType : E_BaseElementType
VAR_INPUT
END_VAR
GetType				:= THIS^.stIdentifier.eType;
END_METHOD

METHOD PUBLIC LinkCommonData : BOOL
VAR_INPUT
	stCommonData				: REFERENCE TO ST_BaseCommonData;
END_VAR
VAR
	bResult						: BOOL;
END_VAR
bResult		:= SUPER^.LinkCommonData (stCommonData := stCommonData);

(* sprawdzenie czy jest podłaczony loger	*)
THIS^.stEvents.bLoggerDataCompleted	:= THIS^.refstCommonData.itfLogger <> 0;

LinkCommonData		:= bResult AND THIS^.stEvents.bLoggerDataCompleted;
END_METHOD

METHOD PUBLIC SetCode
VAR_INPUT
	sCode							: STRING;
	sAdd							: STRING;
END_VAR
THIS^.stIdentifier.sCode				:= sCode;
END_METHOD

(*			
	RafalOS
	Rafał Osajda		03.10.2025		TC 4024.66
	nadawanie unikalnych ID dla zdarzeń
*)
METHOD PUBLIC SetEventsIDs : UINT
VAR_INPUT
	uiNewID		: UINT;
END_VAR
VAR
	uiI			: UINT;
	uitmpValue	: UINT;
	uitmpValue2	: UINT;
END_VAR
IF (THIS^.stEvents.uiNumberOfAdded > 0) THEN
	FOR uiI := 1 TO THIS^.stEvents.uiNumberOfAdded DO
		uitmpValue	:= SEL (uiNewID = 0, uiNewID, 1);
		uitmpValue2	:= uitmpValue + uiI;// - 1;
		THIS^.stEvents.arrDefinitions [uiI].uiIDEvent	:= uitmpValue2;
	END_FOR
	SetEventsIDs				:= uiNewID + THIS^.stEvents.uiNumberOfAdded;
ELSE
	SetEventsIDs				:= uiNewID;
END_IF
END_METHOD

METHOD PUBLIC SetID : UINT
VAR_INPUT
	uiID					: UINT;
END_VAR
THIS^.stIdentifier.uiID			:= uiID;
SetID							:= uiID;
END_METHOD

METHOD PUBLIC SetName
VAR_INPUT
	stName				: ST_BaseLabel;
END_VAR
this^.stIdentifier.stName			:= stName;
END_METHOD

METHOD PUBLIC SetType
VAR_INPUT
	eType					: E_BaseElementType;
END_VAR
THIS^.stIdentifier.eType				:= eType;
END_METHOD

METHOD PUBLIC ZwrocDaneDlaZgloszeniaOID : BOOL
VAR_INPUT
	uiIDZgloszenia				: UINT;
END_VAR
VAR_OUTPUT
	uiIDElementu				: UINT;
	sKodElementu				: STRING;
	sRodzajZgloszenia			: STRING;
	eRodzajZgloszenia			: E_BaseEvents_Category;
	stOpis						: ST_BaseLabel;
	stTekstElementu				: ST_BaseLabel;
END_VAR
VAR
	iI: INT;
END_VAR
FOR iI := 1 TO TO_INT (THIS^.stEvents.uiNumberOfAdded) DO
	IF (THIS^.stEvents.arrDefinitions [iI].uiIDEvent = uiIDElementu) THEN
		uiIDElementu				:= THIS^.stIdentifier.uiID;
	    sKodElementu				:= THIS^.stIdentifier.sCode;
	    sRodzajZgloszenia			:= TO_STRING (THIS^.stEvents.arrDefinitions [iI].eEventCategory);
	    eRodzajZgloszenia			:= THIS^.stEvents.arrDefinitions [iI].eEventCategory;
	    stOpis						:= THIS^.stEvents.arrDefinitions [iI].stDescription;
		stTekstElementu				:= THIS^.stIdentifier.stName;
		ZwrocDaneDlaZgloszeniaOID	:= TRUE;
		EXIT;
	END_IF
END_FOR
END_METHOD

END_FUNCTION_BLOCK

// ---- POUs/A04_FB_BaseComponent/FB_BaseComponent.TcPOU
(*			
	RAFALOS
	Rafał Osajda		19.09.2025		TC 4024.66
	Komponent bazowy dla elementów prostych
*)
FUNCTION_BLOCK FB_BaseComponent EXTENDS FB_BaseLoggerElement IMPLEMENTS ITF_BaseComponent, ITF_BaseComponent_HMI_Connector
VAR
	cmdReset						: FB_BaseCommand;
	cmdParametersCreate				: FB_BaseCommand;
	cmdParametersRestoreToDefault	: FB_BaseCommand;
	
	
END_VAR
VAR PERSISTENT
	stParameters					: ST_Parameters;
END_VAR

(*			
	EVERDE sp. z o.o.
	Rafał Osajda		27.03.2025		TC 4024.66
	Obsluga bledow sprawdzanie czy jakis blad sie nei pojawil i ustawienie stanu lub wylaczenie
*)
METHOD PUBLIC ExecuteEveryCycle_Error
VAR_INPUT
END_VAR
END_METHOD

(*			
	EVERDE sp. z o.o.
	Rafał Osajda		27.03.2025		TC 4024.66
	Wywolanie co cykl operacji 
*)
METHOD PUBLIC ExecuteEveryCycle_Operation
VAR_INPUT
END_VAR
IF (THIS^.cmdReset.OperationExecute ()) THEN
	THIS^.cmdReset.Operation (bIN		:= THIS^.ResetOperation ());
END_IF

IF (THIS^.cmdParametersCreate.OperationExecute ()) THEN
	THIS^.cmdParametersCreate.Operation (bIN := THIS^.ParameterCreateTable ());
END_IF

IF (THIS^.cmdParametersRestoreToDefault.OperationExecute ()) THEN
	THIS^.cmdParametersRestoreToDefault.Operation (bIN	:= THIS^.ParameterRestoreDefaultValueAll ());
END_IF
END_METHOD

(*			
	EVERDE sp. z o.o.
	Rafał Osajda		27.03.2025		TC 4024.66
	Aktualizacja flag 
*)
METHOD PUBLIC ExecuteEveryCycle_Status
VAR_INST
END_VAR
END_METHOD

(*			
	EVERDE sp. z o.o.
	Rafał Osajda		27.03.2025		TC 4024.66
	Testowanie czy nei pojawil sie jakis rozkaz i uruchomienie odpowiednich operacji
*)
METHOD PUBLIC ExecuteEveryCycle_Test
VAR_INPUT
END_VAR
THIS^.cmdReset.Test ();
THIS^.cmdParametersCreate.Test ();
THIS^.cmdParametersRestoreToDefault.Test ();
END_METHOD

METHOD FB_init : BOOL
VAR_INPUT
	bInitRetains : BOOL; // if TRUE, the retain variables are initialized (warm start / cold start)
	bInCopyCode : BOOL;  // if TRUE, the instance afterwards gets moved into the copy code (online change)
END_VAR
THIS^.stIdentifier.eType			:= E_BaseElementType.eComponent;
END_METHOD

(*			
	EVERDE sp. z o.o.
	Rafał Osajda		03.10.2025		TC 4024.66
	
*)
METHOD PUBLIC FirstCycle : BOOL
VAR_INPUT
END_VAR
FirstCycle				:= SUPER^.FirstCycle ();
END_METHOD

METHOD GetITFComponent : ITF_BaseComponent
VAR_INPUT
END_VAR
GetITFComponent		:= THIS^;
END_METHOD

METHOD GetITFControlElement : ITF_BaseControlElement
VAR_INPUT
END_VAR
GetITFControlElement	:= null;
END_METHOD

METHOD GetITFGroupElement : ITF_BaseGroupElement
VAR_INPUT
END_VAR
GetITFGroupElement	:= null;
END_METHOD

METHOD GetITFTopElement : ITF_BaseTopElement
VAR_INPUT
END_VAR
GetITFTopElement		:= null;
END_METHOD

(*			
	EVERDE sp. z o.o.
	Rafał Osajda		07.10.2025		TC 4024.66
	Dodpisywanie się do listy logera
*)
METHOD PUBLIC JoinTheLogger : BOOL
VAR_INPUT
END_VAR
IF (THIS^.bIsValidCommonData) THEN
	IF (THIS^.refstCommonData.itfLogger.AddItem (itfItem := THIS^) > 0 ) THEN
		JoinTheLogger		:= TRUE;
	END_IF
END_IF
END_METHOD

(*			
	EVERDE sp. z o.o.
	Rafał Osajda		26.03.2025		TC 4024.66
	Dodawanie parametru do elementu wykonawczego - metode wywołać przy pierwszym uruchomieniu programu by wgrać parametry do pamięci
	później używać tylko edycji lub przywracania wartości domyślnych
*)
METHOD PUBLIC ParameterAdd : BOOL
VAR_INPUT
	stParameter			: ST_BaseDescriptor;
END_VAR
IF (THIS^.stParameters.uiNumber + 1 <= TO_UINT (GVL_BaseConstans.MAX_NUMBER_OF_PARAMETERS)) THEN
	THIS^.stParameters.uiNumber 		:= THIS^.stParameters.uiNumber + 1;
	THIS^.stParameters.arrRow [THIS^.stParameters.uiNumber] 	:= stParameter;
	ParameterAdd				:= TRUE;
ELSE
	ParameterAdd				:= FALSE;
END_IF
END_METHOD

(*			
	EVERDE sp. z o.o.
	Rafał Osajda		26.03.2025		TC 4024.66
	Modyfikuje wartość domyślną w istniejącym parametrze - true jak się zmiana udała
*)
METHOD PUBLIC ParameterCorrectDefaultValue : BOOL
VAR_INPUT
	uiNumber			: UINT;
	rValue				: REAL;
END_VAR
IF (uiNumber > 0 AND uiNumber <= THIS^.stParameters.uiNumber) THEN
	IF (rValue >= THIS^.GetMinFrom (stIN := THIS^.stParameters.arrRow [uiNumber]) AND
		rValue <= THIS^.GetMaxFrom (stIN := THIS^.stParameters.arrRow [uiNumber])) THEN
		THIS^.SetDefaultValueIn (stIN := THIS^.stParameters.arrRow [uiNumber], rDefaultValue	:= rValue);
		ParameterCorrectDefaultValue		:= TRUE;
	ELSE
		ParameterCorrectDefaultValue		:= FALSE;
	END_IF
ELSE
	ParameterCorrectDefaultValue		:= FALSE;
END_IF
END_METHOD

METHOD PUBLIC ParameterCorrectName : BOOL
VAR_INPUT
	eLocation					: E_BaseLocation;
	uiNumberOfParameter			: UINT;
	wsDescription				: WSTRING;
END_VAR
THIS^.SetTextIn (
	stIN 			:= THIS^.stParameters.arrRow [uiNumberOfParameter],
	eLocation		:= eLocation,
	wsDescription	:= wsDescription
);
END_METHOD

(*			
	EVERDE sp. z o.o.
	Rafał Osajda		26.03.2025		TC 4024.66
	Modyfikuje wartość w istniejącym parametrze - true jak się zmiana udała
*)
METHOD PUBLIC ParameterCorrectValue : BOOL
VAR_INPUT
	uiNumber			: UINT;
	rValue				: REAL;
END_VAR
IF (uiNumber > 0 AND uiNumber <= THIS^.stParameters.uiNumber) THEN
	IF (rValue <= THIS^.GetMaxFrom (stIN := THIS^.stParameters.arrRow [uiNumber]) AND
		rValue >= THIS^.GetMinFrom (stIN := THIS^.stParameters.arrRow [uiNumber]) ) THEN
		THIS^.SetValueIn (
			stIN		:= THIS^.stParameters.arrRow [uiNumber],
			rValue		:= rValue
		);
		ParameterCorrectValue		:= TRUE;
	ELSE
		ParameterCorrectValue		:= FALSE;
	END_IF
ELSE
	ParameterCorrectValue		:= FALSE;
END_IF
END_METHOD

(*			
	EVERDE sp. z o.o.
	Rafał Osajda		31.03.2025		TC 4024.66
	Metoda wymazująca dotychczasowe dane z tablicy parametrów i przypisująca je od nowa
*)
METHOD PROTECTED ParameterCreateTable : BOOL
VAR_INPUT
END_VAR
MEMSET (
	destAddr			:= ADR (THIS^.stParameters.arrRow),
	fillByte			:= 0,
	n					:= SIZEOF (THIS^.stParameters.arrRow)
);
THIS^.stParameters.uiNumber	:= 0;

ParameterCreateTable := TRUE;
END_METHOD

METHOD PUBLIC ParameterGet : ST_BaseDescriptor
VAR_INPUT
	uiNumer				: UINT;
END_VAR
ParameterGet			:= THIS^.stParameters.arrRow [uiNumer];
END_METHOD

(*			
	EVERDE sp. z o.o.
	Rafał Osajda		26.03.2025		TC 4024.66
	Zwraca wartosc domyslna
*)
METHOD PUBLIC ParameterGetDefaultValue : REAL
VAR_INPUT
	uiNumber				: UINT;
END_VAR
IF (uiNumber > 0 AND uiNumber <= THIS^.stParameters.uiNumber) THEN
	ParameterGetDefaultValue			:= THIS^.GetDefaultValueFrom (stIN :=  THIS^.stParameters.arrRow [uiNumber]);
ELSE
	ParameterGetDefaultValue			:= 0;
END_IF
END_METHOD

(*			
	EVERDE sp. z o.o.
	Rafał Osajda		26.03.2025		TC 4024.66
	Zwraca wartość MAX
*)
METHOD PUBLIC ParameterGetMax : REAL
VAR_INPUT
	uiNumber				: UINT;
END_VAR
IF (uiNumber > 0 AND uiNumber <= THIS^.stParameters.uiNumber) THEN
	ParameterGetMax			:= THIS^.GetMaxFrom (stIN :=  THIS^.stParameters.arrRow [uiNumber]);
ELSE
	ParameterGetMax			:= 0;
END_IF
END_METHOD

(*			
	EVERDE sp. z o.o.
	Rafał Osajda		26.03.2025		TC 4024.66
	Zwraca wartość MIN
*)
METHOD PUBLIC ParameterGetMin : REAL
VAR_INPUT
	uiNumber				: UINT;
END_VAR
IF (uiNumber >= 0 AND uiNumber <= THIS^.stParameters.uiNumber) THEN
	ParameterGetMin			:= THIS^.GetMinFrom (stIN := THIS^.stParameters.arrRow [uiNumber]);
ELSE
	ParameterGetMin			:= 0;
END_IF
END_METHOD

METHOD PUBLIC ParameterGetNumberOfAdded : UINT
VAR_INPUT
END_VAR
ParameterGetNumberOfAdded			:= THIS^.stParameters.uiNumber;
END_METHOD

(*			
	EVERDE sp. z o.o.
	Rafał Osajda		26.03.2025		TC 4024.66
	Zwraca jednostke
*)
METHOD PUBLIC ParameterGetUnit : STRING(6)
VAR_INPUT
	uiNumber				: uINT;
END_VAR
IF (uiNumber > 0 AND uiNumber <= THIS^.stParameters.uiNumber) THEN
	ParameterGetUnit			:= THIS^.GetUnitFrom (stIN :=  THIS^.stParameters.arrRow [uiNumber]);
ELSE
	ParameterGetUnit			:= '';
END_IF
END_METHOD

(*			
	EVERDE sp. z o.o.
	Rafał Osajda		26.03.2025		TC 4024.66
	Zwraca wartość
*)
METHOD PUBLIC ParameterGetValue : REAL
VAR_INPUT
	uiNumber				: UINT;
END_VAR
IF (uiNumber > 0 AND uiNumber <= THIS^.stParameters.uiNumber) THEN
	ParameterGetValue			:= THIS^.GetValueFrom (stIN := THIS^.stParameters.arrRow [uiNumber]);
ELSE
	ParameterGetValue			:= 0;
END_IF
END_METHOD

(*			
	EVERDE sp. z o.o.
	Rafał Osajda		26.03.2025		TC 4024.66
	Modyfikacja istniejącego parametra jako przypisanie nowego deskryptora
*)
METHOD PUBLIC ParameterModify : BOOL
VAR_INPUT
	uiNumber			: UINT;
	stParameter			: ST_BaseDescriptor;
END_VAR
IF (uiNumber > 0 AND uiNumber <= THIS^.stParameters.uiNumber) THEN
	THIS^.stParameters.arrRow [uiNumber]	:= 	stParameter;
	ParameterModify		:= TRUE;
ELSE
	ParameterModify		:= FALSE;
END_IF
END_METHOD

METHOD PUBLIC ParameterRestoreDefaultValue : BOOL
VAR_INPUT
	uiNumber		: UINT;
END_VAR
IF (uiNumber > 0 AND uiNumber <= THIS^.stParameters.uiNumber) THEN
	THIS^.SetValueIn (stIN := THIS^.stParameters.arrRow [uiNumber], rValue := THIS^.GetDefaultValueFrom (stIN := THIS^.stParameters.arrRow [uiNumber]));
	ParameterRestoreDefaultValue	:= TRUE;
ELSE
	ParameterRestoreDefaultValue	:= FALSE;
END_IF
END_METHOD

METHOD PROTECTED ParameterRestoreDefaultValueAll : BOOL
VAR_INPUT
END_VAR

VAR
	iI					: INT;
	bResult				: bool;
END_VAR
bResult					:= TRUE;
FOR iI := 1 TO TO_INT (THIS^.stParameters.uiNumber) DO 
	bResult				:= bResult AND THIS^.ParameterRestoreDefaultValue (uiNumber := TO_UINT (iI));
END_FOR
END_METHOD

(*			
	EVERDE sp. z o.o.
	Rafał Osajda		04.05.2025		TC 4024.66
	Skasowanie i utworzenie tablicy parametrów od nowa 
*)
METHOD PUBLIC ParametersCreate : BOOL
THIS^.cmdParametersCreate.Execute ();
END_METHOD

(*			
	EVERDE sp. z o.o.
	Rafał Osajda		04.05.2025		TC 4024.66
	Przywrocenie parametrow - in na false to tylko ten element true razem z podelementami
*)
METHOD PUBLIC ParameterSetToDefault : BOOL
THIS^.cmdParametersRestoreToDefault.Execute ();
END_METHOD

METHOD PUBLIC Reset : BOOL
VAR_INPUT
END_VAR
THIS^.cmdReset.Execute ();
END_METHOD

METHOD PUBLIC ResetGetBusy : BOOL
VAR_INPUT
END_VAR
ResetGetBusy		:= THIS^.cmdReset.IsBusy ();
END_METHOD

METHOD PUBLIC ResetGetStatus : BOOL
VAR_INPUT
END_VAR
ResetGetStatus			:= THIS^.cmdReset.IsStatus ();
END_METHOD

METHOD PROTECTED ResetOperation : BOOL
VAR_INPUT
END_VAR


ResetOperation			:= FALSE;
END_METHOD

END_FUNCTION_BLOCK

// ---- POUs/A05_FB_BaseControlElement/FB_BaseControlElement.TcPOU
(*			
	RAFALOS
	Rafał Osajda		19.09.2025		TC 4024.66
	Rodzic dla wszystkich elementów wykonawczych
*)
FUNCTION_BLOCK FB_BaseControlElement EXTENDS FB_BaseComponent IMPLEMENTS ITF_BaseControlElement, ITF_BaseControlElement_HMI_Connector
VAR
	arrComponent			: ARRAY  [1..GVL_BaseConstans.MAX_ITEM_PER_ELEMENT] OF ITF_BaseComponent;
	uiNumberOfComponents	: UINT;
(*	Zasilanie	*)
	itfSS1					: ITF_BaseFlagGet;
	itfSTO					: ITF_BaseFlagGet;
	stPower					: ST_BaseControlElement_Power;
(*	Bazowanie	*)
	stHoming				: ST_BaseControlElement_Homing;
(*	Flagi główne elementów	*)
	bPosition0				: BOOL := TRUE;	//jak nie potrzebna to zostawić na true w przeciwnym przypadku przypisać odpowiednią logikę
	bDoNothing				: BOOL := TRUE;	//jak nie potrzebna to zostawić na true w przeciwnym przypadku przypisać odpowiednią logikę
	
END_VAR

METHOD PROTECTED AddComponent : BOOL
VAR_INPUT
	itfComponent				: ITF_BaseComponent;
END_VAR
IF (THIS^.uiNumberOfComponents + 1 <= GVL_BaseConstans.MAX_ITEM_PER_ELEMENT) THEN
	THIS^.uiNumberOfComponents		:= THIS^.uiNumberOfComponents + 1;
	THIS^.arrComponent [THIS^.uiNumberOfComponents]	:= itfComponent;
	AddComponent				:= TRUE;
ELSE
	;//zwrocenie zbyt dużo komponentow
END_IF
END_METHOD

(*			
	EVERDE sp. z o.o.
	Rafał Osajda		24.03.2025		TC 4024.66
	Definicja nowego zgłoszenia
*)
METHOD PUBLIC EventsDefinition : BOOL
SUPER^.EventsDefinition ();

THIS^.SetText (eLocation := E_BaseLocation.pl, wsDescription	:= "Błąd uruchomienia zasilania - brak zgody od safety - BRAK SS1");
THIS^.SetText (eLocation := E_BaseLocation.en, wsDescription	:= "");
THIS^.SetText (eLocation := E_BaseLocation.de, wsDescription	:= "");
THIS^.AddEvent (
	bIgnoreRepetitions			:= TRUE,
	eEventCategory				:= E_BaseEvents_Category.Error,
	bConfirm					:= FALSE,
	stDescription				:= THIS^.GetTexts ()
);
THIS^.SetText (eLocation := E_BaseLocation.pl, wsDescription	:= "Błąd uruchomienia zasilania - brak zgody od safety - BRAK STO");
THIS^.SetText (eLocation := E_BaseLocation.en, wsDescription	:= "");
THIS^.SetText (eLocation := E_BaseLocation.de, wsDescription	:= "");
THIS^.AddEvent (
	bIgnoreRepetitions			:= TRUE,
	eEventCategory				:= E_BaseEvents_Category.Error,
	bConfirm					:= FALSE,
	stDescription				:= THIS^.GetTexts ()
);
END_METHOD

(*			
	EVERDE sp. z o.o.
	Rafał Osajda		27.03.2025		TC 4024.66
	Obsluga bledow sprawdzanie czy jakis blad sie nei pojawil i ustawienie stanu lub wylaczenie
*)
METHOD PUBLIC ExecuteEveryCycle_Error
VAR
	iI				: INT;
END_VAR
SUPER^.ExecuteEveryCycle_Error ();

FOR iI := 1 TO TO_INT (THIS^.uiNumberOfComponents) DO
	THIS^.arrComponent [iI].ExecuteEveryCycle_Error ();
END_FOR
END_METHOD

(*			
	EVERDE sp. z o.o.
	Rafał Osajda		27.03.2025		TC 4024.66
	Wywolanie co cykl operacji 
*)
METHOD PUBLIC ExecuteEveryCycle_Operation
VAR
	iI			: INT;
	bError		: BOOL;
END_VAR
SUPER^.ExecuteEveryCycle_Operation ();

FOR iI := 1 TO TO_INT (THIS^.uiNumberOfComponents) DO
	THIS^.arrComponent [iI].ExecuteEveryCycle_Operation ();
END_FOR


(* 	Zasilanie	*)
IF (THIS^.stPower.cmdTurnOn.OperationExecute ()) THEN
	bError				:= FALSE;
	IF (NOT THIS^.itfSS1.GetFlag ()) THEN
		//blad 
		THIS^.EventSetActive (iNumber := 1);
		bError			:= TRUE;
	END_IF
	IF (NOT THIS^.itfSTO.GetFlag ()) THEN
		//blad
		THIS^.EventSetActive (iNumber := 2);
		bError			:= TRUE;
	END_IF
	IF (NOT bError) THEN
		THIS^.stPower.cmdTurnOn.Operation (bIN		:= THIS^.PowerOnCycle ());
		IF (THIS^.EventIsActive (iNumber := 1)) THEN
			THIS^.EventSetInactive (iNumber := 1);
		END_IF
		IF (THIS^.EventIsActive (iNumber := 2)) THEN
			THIS^.EventSetInactive (iNumber := 2);
		END_IF
	ELSE
		THIS^.stPower.cmdTurnOn.Abort ();
	END_IF
END_IF
IF (THIS^.stPower.cmdTurnOff.OperationExecute ()) THEN
	THIS^.stPower.cmdTurnOff.Operation (bIN	:= THIS^.PowerOffCycle ());
END_IF
(*	Bazowanie	*)
IF (THIS^.stHoming.cmdExecute.OperationExecute ()) THEN
	THIS^.stHoming.cmdExecute.Operation (bIN	:= THIS^.HomingCycleInternal ());
END_IF
END_METHOD

(*			
	EVERDE sp. z o.o.
	Rafał Osajda		27.03.2025		TC 4024.66
	Aktualizacja flag 
*)
METHOD PUBLIC ExecuteEveryCycle_Status
VAR
	iI				: INT;
END_VAR
SUPER^.ExecuteEveryCycle_Status ();

FOR iI := 1 TO TO_INT (THIS^.uiNumberOfComponents) DO
	THIS^.arrComponent [iI].ExecuteEveryCycle_Status ();
END_FOR
END_METHOD

(*			
	EVERDE sp. z o.o.
	Rafał Osajda		27.03.2025		TC 4024.66
	Testowanie czy nei pojawil sie jakis rozkaz i uruchomienie odpowiednich operacji
*)
METHOD PUBLIC ExecuteEveryCycle_Test
VAR
	iI				: INT;
END_VAR
SUPER^.ExecuteEveryCycle_Test ();

FOR iI := 1 TO TO_INT (THIS^.uiNumberOfComponents) DO
	THIS^.arrComponent [iI].ExecuteEveryCycle_Test ();
END_FOR

THIS^.stPower.cmdTurnOn.Test ();
THIS^.stPower.cmdTurnOff.Test ();

IF (THIS^.stPower.bStatus) THEN
	THIS^.ExecuteEveryCycle_TestWithPower ();
ELSE
	THIS^.ExecuteEveryCycle_TestWithoutPower ();
END_IF
END_METHOD

METHOD PROTECTED ExecuteEveryCycle_TestWithoutPower
VAR_INPUT
END_VAR
THIS^.stHoming.cmdExecute.Abort ();
END_METHOD

METHOD PROTECTED ExecuteEveryCycle_TestWithPower
VAR_INPUT
END_VAR
THIS^.stHoming.cmdExecute.Test ();
END_METHOD

METHOD FB_init : BOOL
VAR_INPUT
	bInitRetains : BOOL; // if TRUE, the retain variables are initialized (warm start / cold start)
	bInCopyCode : BOOL;  // if TRUE, the instance afterwards gets moved into the copy code (online change)
END_VAR
THIS^.stIdentifier.eType			:= E_BaseElementType.eControl;
END_METHOD

METHOD PUBLIC FirstCycle : BOOL
VAR_INPUT
END_VAR
VAR
	bResult			: bool;
	iI				: INT;
END_VAR
bResult				:= SUPER^.FirstCycle ();

FOR iI := 1 TO TO_INT (THIS^.uiNumberOfComponents) DO
	bResult			:= bResult AND THIS^.arrComponent [iI].FirstCycle ();
END_FOR

FirstCycle			:= bResult;
END_METHOD

METHOD GetITFControlElement : ITF_BaseControlElement
VAR_INPUT
END_VAR
GetITFControlElement	:= THIS^;
END_METHOD

METHOD GetITFGroupElement : ITF_BaseGroupElement
VAR_INPUT
END_VAR
GetITFGroupElement	:= null;
END_METHOD

METHOD GetITFTopElement : ITF_BaseTopElement
VAR_INPUT
END_VAR
GetITFTopElement		:= null;
END_METHOD

(*			
	EVERDE sp. z o.o.
	Rafał Osajda		27.05.2025		TC 4024.66
	Metoda bazowania kontrektnego elementu 
*)
METHOD PROTECTED HomingCycle : BOOL
VAR_INPUT
END_VAR
HomingCycle					:= FALSE;
END_METHOD

